      A     M    163.3;
      =     L      4.0;
      BLD   103;
      A     M     21.0;
      =     L      4.1;
      BLD   103;
      A     M     20.1;
      =     L      4.2;
      BLD   103;
      A     M     20.1;
      =     L      4.3;
      BLD   103;
      A     I      8.7;
      =     L      4.4;
      BLD   103;
      A     M     20.0;
      =     L      4.5;
      BLD   103;
      A     M    163.1;
      =     L      4.6;
      BLD   103;
      A     M    163.2;
      =     L      4.7;
      BLD   103;
      CALL FC   180 (
           IN0                      := L      4.0,
           IN1                      := L      4.1,
           IN2                      := L      4.2,
           IN3                      := L      4.3,
           IN4                      := L      4.4,
           IN5                      := L      4.5,
           IN6                      := L      4.6,
           IN7                      := L      4.7,
           IN8                      := W#16#2,
           IN9                      := C      9,
           OUT10                    := DB10.DBW   26,
           OUT11                    := Q      6.3,
           OUT12                    := M    163.4,
           OUT13                    := M    163.5,
           IO14                     := DB181.DBW   18,
           IO15                     := DB10.DBW   60);
      NOP   0;
NETWORK
TITLE =

      A     I      8.7;
      =     L      4.0;
      A     L      4.0;
      BLD   102;
      =     Q      3.6;
      O     L      4.0;
      O     I      1.3;
      =     Q      4.5;
END_FUNCTION

FUNCTION FC 15 : VOID
AUTHOR :
FAMILY : DRIVES
NAME : DRIVES
VERSION : 0.1


VAR_TEMP
  TEMP0 : REAL ;
END_VAR
BEGIN
NETWORK
TITLE =

      A     I      0.2;
      AN    M    164.4;
      A(    ;
      A(    ;
      O     Q      0.0;
      O     I      1.0;
      O     I      2.0;
      O     I      2.2;
      O     I      2.3;
      O     I      2.4;
      O     I      2.6;
      O     I      2.7;
      O(    ;
      A     I      4.1;
      FP    M    218.1;
      )     ;
      )     ;
      =     M    218.0;
      A     M    218.0;
      )     ;
      FP    M    164.0;
      =     M    164.1;
NETWORK
TITLE =

      A(    ;
      A     M     38.0;
      A(    ;
      O     I     11.4;
      O     I     12.5;
      )     ;
      L     DB2.DBW   54;
      SD    T     27;
      NOP   0;
      NOP   0;
      NOP   0;
      A     T     27;
      )     ;
      FP    M    218.3;
      =     M    164.2;
NETWORK
TITLE =
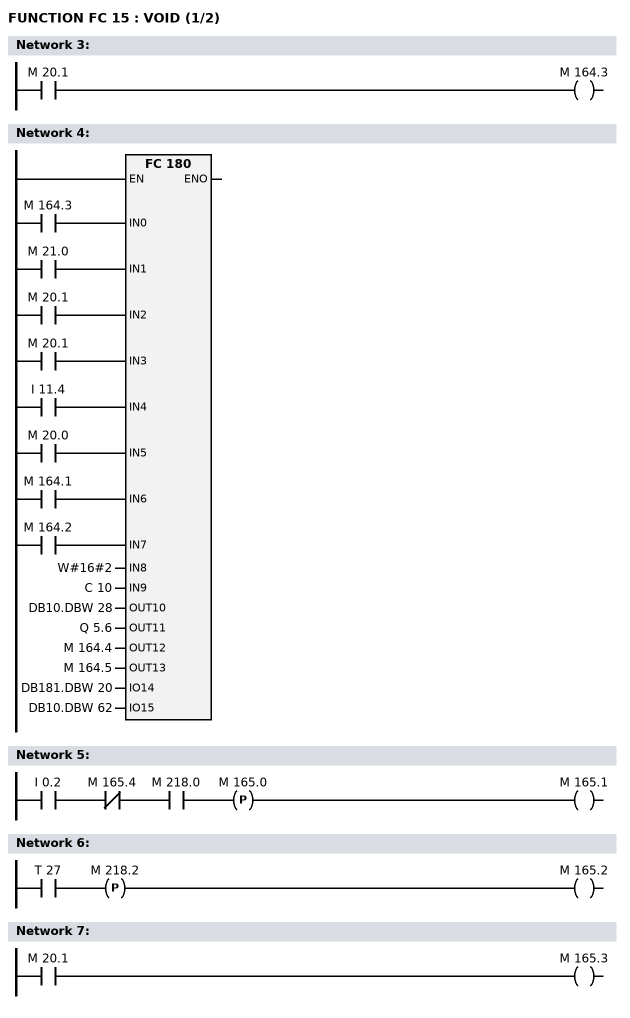

      A     M     20.1;
      =     M    164.3;
NETWORK
TITLE =

      A     M    164.3;
      =     L      4.0;
      BLD   103;
      A     M     21.0;
      =     L      4.1;
      BLD   103;
      A     M     20.1;
      =     L      4.2;
      BLD   103;
      A     M     20.1;
      =     L      4.3;
      BLD   103;
      A     I     11.4;
      =     L      4.4;
      BLD   103;
      A     M     20.0;
      =     L      4.5;
      BLD   103;
      A     M    164.1;
      =     L      4.6;
      BLD   103;
      A     M    164.2;
      =     L      4.7;
      BLD   103;
      CALL FC   180 (
           IN0                      := L      4.0,
           IN1                      := L      4.1,
           IN2                      := L      4.2,
           IN3                      := L      4.3,
           IN4                      := L      4.4,
           IN5                      := L      4.5,
           IN6                      := L      4.6,
           IN7                      := L      4.7,
           IN8                      := W#16#2,
           IN9                      := C     10,
           OUT10                    := DB10.DBW   28,
           OUT11                    := Q      5.6,
           OUT12                    := M    164.4,
           OUT13                    := M    164.5,
           IO14                     := DB181.DBW   20,
           IO15                     := DB10.DBW   62);
      NOP   0;
NETWORK
TITLE =

      A     I      0.2;
      AN    M    165.4;
      A     M    218.0;
      FP    M    165.0;
      =     M    165.1;
NETWORK
TITLE =

      A     T     27;
      FP    M    218.2;
      =     M    165.2;
NETWORK
TITLE =

      A     M     20.1;
      =     M    165.3;
NETWORK
TITLE =
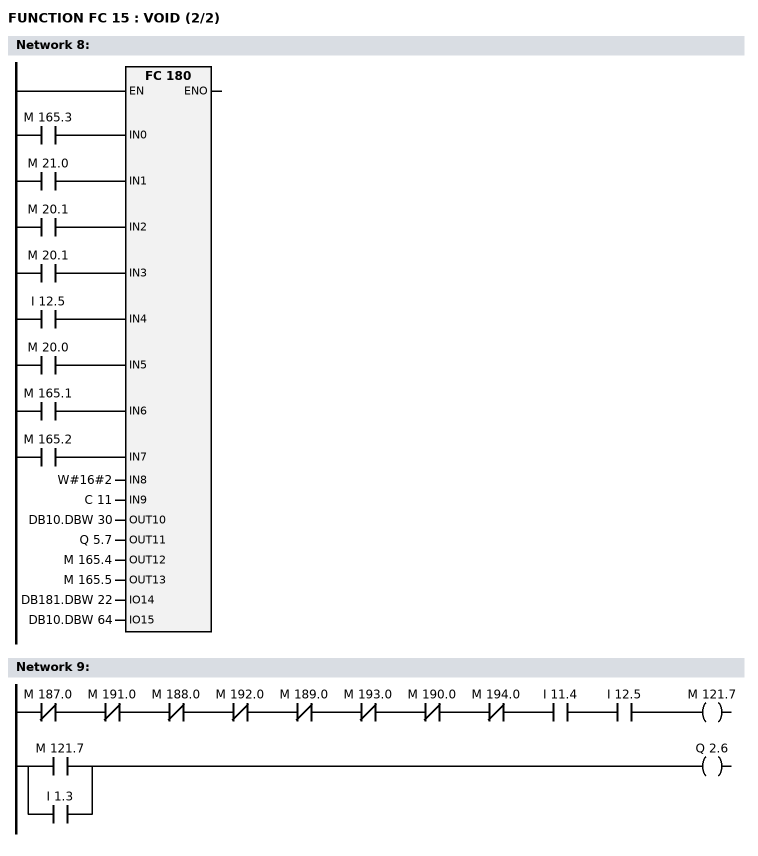

      A     M    165.3;
      =     L      4.0;
      BLD   103;
      A     M     21.0;
      =     L      4.1;
      BLD   103;
      A     M     20.1;
      =     L      4.2;
      BLD   103;
      A     M     20.1;
      =     L      4.3;
      BLD   103;
      A     I     12.5;
      =     L      4.4;
      BLD   103;
      A     M     20.0;
      =     L      4.5;
      BLD   103;
      A     M    165.1;
      =     L      4.6;
      BLD   103;
      A     M    165.2;
      =     L      4.7;
      BLD   103;
      CALL FC   180 (
           IN0                      := L      4.0,
           IN1                      := L      4.1,
           IN2                      := L      4.2,
           IN3                      := L      4.3,
           IN4                      := L      4.4,
           IN5                      := L      4.5,
           IN6                      := L      4.6,
           IN7                      := L      4.7,
           IN8                      := W#16#2,
           IN9                      := C     11,
           OUT10                    := DB10.DBW   30,
           OUT11                    := Q      5.7,
           OUT12                    := M    165.4,
           OUT13                    := M    165.5,
           IO14                     := DB181.DBW   22,
           IO15                     := DB10.DBW   64);
      NOP   0;
NETWORK
TITLE =

      AN    M    187.0;
      AN    M    191.0;
      AN    M    188.0;
      AN    M    192.0;
      AN    M    189.0;
      AN    M    193.0;
      AN    M    190.0;
      AN    M    194.0;
      A     I     11.4;
      A     I     12.5;
      =     M    121.7;
      A     M    121.7;
      O     I      1.3;
      =     Q      2.6;
END_FUNCTION

FUNCTION FC 20 : VOID
AUTHOR :
FAMILY : ANALOGUE
NAME : ANALOGUE
VERSION : 0.1


VAR_TEMP
  TEMP0 : WORD ;
  TEMP1 : REAL ;
  TEMP2 : REAL ;
  TEMP3 : REAL ;
END_VAR
BEGIN
NETWORK
TITLE =
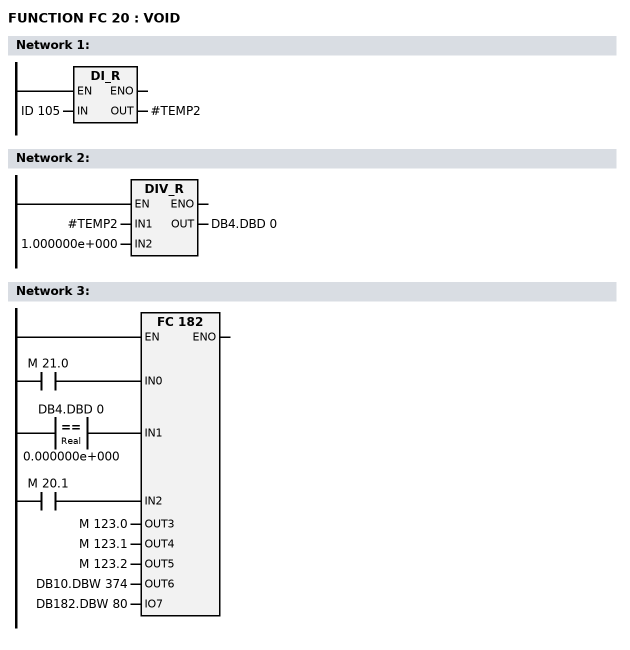

      L     ID   105;
      DTR   ;
      T     #TEMP2;
      NOP   0;
NETWORK
TITLE =

      L     #TEMP2;
      L     1.000000e+000;
      /R    ;
      T     DB4.DBD    0;
      NOP   0;
NETWORK
TITLE =

      A     M     21.0;
      =     L     14.0;
      BLD   103;
      A(    ;
      L     DB4.DBD    0;
      L     0.000000e+000;
      ==R   ;
      )     ;
      =     L     14.1;
      BLD   103;
      A     M     20.1;
      =     L     14.2;
      BLD   103;
      CALL FC   182 (
           IN0                      := L     14.0,
           IN1                      := L     14.1,
           IN2                      := L     14.2,
           OUT3                     := M    123.0,
           OUT4                     := M    123.1,
           OUT5                     := M    123.2,
           OUT6                     := DB10.DBW  374,
           IO7                      := DB182.DBW   80);
      NOP   0;
NETWORK
TITLE =

      A     M    200.6;
      A     M     20.1;
      =     L     14.0;
      A     L     14.0;
      JNB   M001;
      L     DW#16#80000000;
      T     QD   105;
M001: NOP   0;
      AN    L     14.0;
      JNB   M002;
      L     DW#16#0;
      T     QD   105;
M002: NOP   0;
NETWORK
TITLE =

      L     DB4.DBD    0;
      L     DB4.DBD    4;
      >=R   ;
      =     M    116.0;
      =     Q      4.1;
NETWORK
TITLE =

      A(    ;
      L     DB4.DBD    0;
      L     DB4.DBD   12;
      >=R   ;
      )     ;
      A(    ;
      A(    ;
      O     M    116.3;
      O     M    116.5;
      )     ;
      FP    M    122.0;
      )     ;
      S     M    122.1;
      A     Q      6.6;
      R     M    122.1;
      A     M    122.1;
      =     L     14.0;
      A     L     14.0;
      BLD   102;
      =     Q      3.7;
      O     L     14.0;
      O     I      1.3;
      =     Q      1.4;
NETWORK
TITLE =
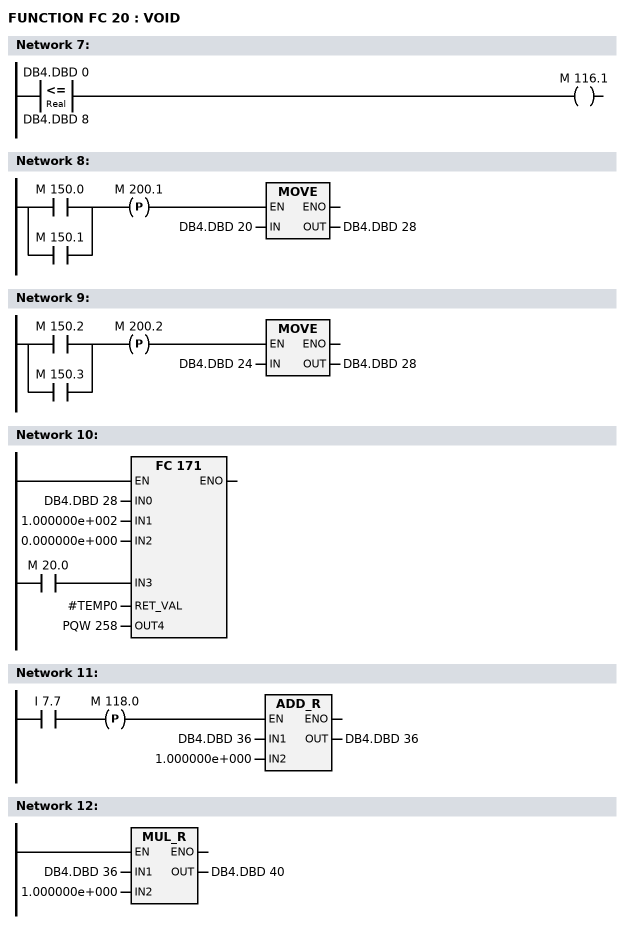

      L     DB4.DBD    0;
      L     DB4.DBD    8;
      <=R   ;
      =     M    116.1;
NETWORK
TITLE =

      A(    ;
      O     M    150.0;
      O     M    150.1;
      )     ;
      FP    M    200.1;
      JNB   M003;
      L     DB4.DBD   20;
      T     DB4.DBD   28;
M003: NOP   0;
NETWORK
TITLE =

      A(    ;
      O     M    150.2;
      O     M    150.3;
      )     ;
      FP    M    200.2;
      JNB   M004;
      L     DB4.DBD   24;
      T     DB4.DBD   28;
M004: NOP   0;
NETWORK
TITLE =

      A     M     20.0;
      =     L     14.0;
      BLD   103;
      CALL FC   171 (
           IN0                      := DB4.DBD   28,
           IN1                      := 1.000000e+002,
           IN2                      := 0.000000e+000,
           IN3                      := L     14.0,
           RET_VAL                  := #TEMP0,
           OUT4                     := PQW  258);
      NOP   0;
NETWORK
TITLE =

      A     I      7.7;
      FP    M    118.0;
      JNB   M005;
      L     DB4.DBD   36;
      L     1.000000e+000;
      +R    ;
      T     DB4.DBD   36;
M005: NOP   0;
NETWORK
TITLE =

      L     DB4.DBD   36;
      L     1.000000e+000;
      *R    ;
      T     DB4.DBD   40;
      NOP   0;
NETWORK
TITLE =

      A(    ;
      A(    ;
      A     M    151.3;
      L     DB2.DBW   40;
      SF    T     20;
      NOP   0;
      NOP   0;
      NOP   0;
      A     T     20;
      )     ;
      A(    ;
      O     M    116.5;
      O     M    116.2;
      )     ;
      O     ;
      A(    ;
      A     M    151.2;
      L     DB2.DBW   42;
      SF    T     21;
      NOP   0;
      NOP   0;
      NOP   0;
      A     T     21;
      )     ;
      A(    ;
      O     M    116.3;
      O     M    116.6;
      )     ;
      )     ;
      FP    M    118.2;
      JNB   M006;
      L     0.000000e+000;
      T     DB4.DBD   36;
M006: NOP   0;
NETWORK
TITLE =
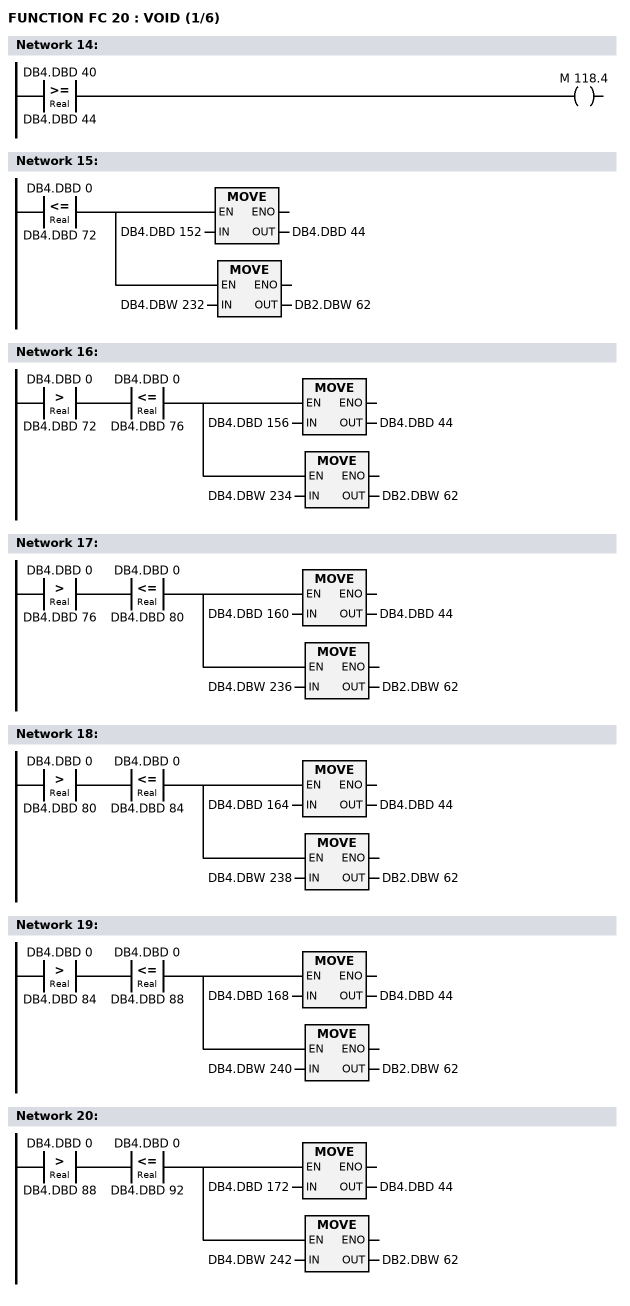

      L     DB4.DBD   40;
      L     DB4.DBD   44;
      >=R   ;
      =     M    118.4;
NETWORK
TITLE =

      L     DB4.DBD    0;
      L     DB4.DBD   72;
      <=R   ;
      =     L     14.0;
      A     L     14.0;
      JNB   M007;
      L     DB4.DBD  152;
      T     DB4.DBD   44;
M007: NOP   0;
      A     L     14.0;
      JNB   M008;
      L     DB4.DBW  232;
      T     DB2.DBW   62;
M008: NOP   0;
NETWORK
TITLE =

      A(    ;
      L     DB4.DBD    0;
      L     DB4.DBD   72;
      >R    ;
      )     ;
      A(    ;
      L     DB4.DBD    0;
      L     DB4.DBD   76;
      <=R   ;
      )     ;
      =     L     14.0;
      A     L     14.0;
      JNB   M009;
      L     DB4.DBD  156;
      T     DB4.DBD   44;
M009: NOP   0;
      A     L     14.0;
      JNB   M00a;
      L     DB4.DBW  234;
      T     DB2.DBW   62;
M00a: NOP   0;
NETWORK
TITLE =

      A(    ;
      L     DB4.DBD    0;
      L     DB4.DBD   76;
      >R    ;
      )     ;
      A(    ;
      L     DB4.DBD    0;
      L     DB4.DBD   80;
      <=R   ;
      )     ;
      =     L     14.0;
      A     L     14.0;
      JNB   M00b;
      L     DB4.DBD  160;
      T     DB4.DBD   44;
M00b: NOP   0;
      A     L     14.0;
      JNB   M00c;
      L     DB4.DBW  236;
      T     DB2.DBW   62;
M00c: NOP   0;
NETWORK
TITLE =

      A(    ;
      L     DB4.DBD    0;
      L     DB4.DBD   80;
      >R    ;
      )     ;
      A(    ;
      L     DB4.DBD    0;
      L     DB4.DBD   84;
      <=R   ;
      )     ;
      =     L     14.0;
      A     L     14.0;
      JNB   M00d;
      L     DB4.DBD  164;
      T     DB4.DBD   44;
M00d: NOP   0;
      A     L     14.0;
      JNB   M00e;
      L     DB4.DBW  238;
      T     DB2.DBW   62;
M00e: NOP   0;
NETWORK
TITLE =

      A(    ;
      L     DB4.DBD    0;
      L     DB4.DBD   84;
      >R    ;
      )     ;
      A(    ;
      L     DB4.DBD    0;
      L     DB4.DBD   88;
      <=R   ;
      )     ;
      =     L     14.0;
      A     L     14.0;
      JNB   M00f;
      L     DB4.DBD  168;
      T     DB4.DBD   44;
M00f: NOP   0;
      A     L     14.0;
      JNB   M010;
      L     DB4.DBW  240;
      T     DB2.DBW   62;
M010: NOP   0;
NETWORK
TITLE =

      A(    ;
      L     DB4.DBD    0;
      L     DB4.DBD   88;
      >R    ;
      )     ;
      A(    ;
      L     DB4.DBD    0;
      L     DB4.DBD   92;
      <=R   ;
      )     ;
      =     L     14.0;
      A     L     14.0;
      JNB   M011;
      L     DB4.DBD  172;
      T     DB4.DBD   44;
M011: NOP   0;
      A     L     14.0;
      JNB   M012;
      L     DB4.DBW  242;
      T     DB2.DBW   62;
M012: NOP   0;
NETWORK
TITLE =
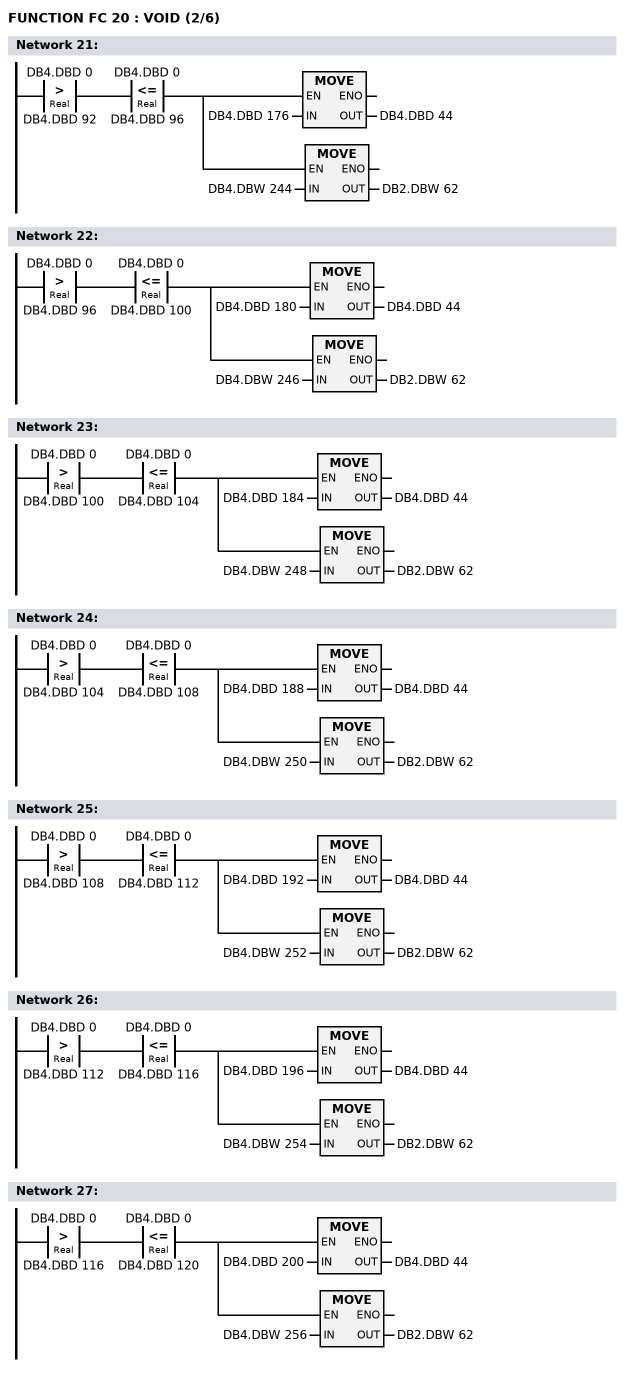

      A(    ;
      L     DB4.DBD    0;
      L     DB4.DBD   92;
      >R    ;
      )     ;
      A(    ;
      L     DB4.DBD    0;
      L     DB4.DBD   96;
      <=R   ;
      )     ;
      =     L     14.0;
      A     L     14.0;
      JNB   M013;
      L     DB4.DBD  176;
      T     DB4.DBD   44;
M013: NOP   0;
      A     L     14.0;
      JNB   M014;
      L     DB4.DBW  244;
      T     DB2.DBW   62;
M014: NOP   0;
NETWORK
TITLE =

      A(    ;
      L     DB4.DBD    0;
      L     DB4.DBD   96;
      >R    ;
      )     ;
      A(    ;
      L     DB4.DBD    0;
      L     DB4.DBD  100;
      <=R   ;
      )     ;
      =     L     14.0;
      A     L     14.0;
      JNB   M015;
      L     DB4.DBD  180;
      T     DB4.DBD   44;
M015: NOP   0;
      A     L     14.0;
      JNB   M016;
      L     DB4.DBW  246;
      T     DB2.DBW   62;
M016: NOP   0;
NETWORK
TITLE =

      A(    ;
      L     DB4.DBD    0;
      L     DB4.DBD  100;
      >R    ;
      )     ;
      A(    ;
      L     DB4.DBD    0;
      L     DB4.DBD  104;
      <=R   ;
      )     ;
      =     L     14.0;
      A     L     14.0;
      JNB   M017;
      L     DB4.DBD  184;
      T     DB4.DBD   44;
M017: NOP   0;
      A     L     14.0;
      JNB   M018;
      L     DB4.DBW  248;
      T     DB2.DBW   62;
M018: NOP   0;
NETWORK
TITLE =

      A(    ;
      L     DB4.DBD    0;
      L     DB4.DBD  104;
      >R    ;
      )     ;
      A(    ;
      L     DB4.DBD    0;
      L     DB4.DBD  108;
      <=R   ;
      )     ;
      =     L     14.0;
      A     L     14.0;
      JNB   M019;
      L     DB4.DBD  188;
      T     DB4.DBD   44;
M019: NOP   0;
      A     L     14.0;
      JNB   M01a;
      L     DB4.DBW  250;
      T     DB2.DBW   62;
M01a: NOP   0;
NETWORK
TITLE =

      A(    ;
      L     DB4.DBD    0;
      L     DB4.DBD  108;
      >R    ;
      )     ;
      A(    ;
      L     DB4.DBD    0;
      L     DB4.DBD  112;
      <=R   ;
      )     ;
      =     L     14.0;
      A     L     14.0;
      JNB   M01b;
      L     DB4.DBD  192;
      T     DB4.DBD   44;
M01b: NOP   0;
      A     L     14.0;
      JNB   M01c;
      L     DB4.DBW  252;
      T     DB2.DBW   62;
M01c: NOP   0;
NETWORK
TITLE =

      A(    ;
      L     DB4.DBD    0;
      L     DB4.DBD  112;
      >R    ;
      )     ;
      A(    ;
      L     DB4.DBD    0;
      L     DB4.DBD  116;
      <=R   ;
      )     ;
      =     L     14.0;
      A     L     14.0;
      JNB   M01d;
      L     DB4.DBD  196;
      T     DB4.DBD   44;
M01d: NOP   0;
      A     L     14.0;
      JNB   M01e;
      L     DB4.DBW  254;
      T     DB2.DBW   62;
M01e: NOP   0;
NETWORK
TITLE =

      A(    ;
      L     DB4.DBD    0;
      L     DB4.DBD  116;
      >R    ;
      )     ;
      A(    ;
      L     DB4.DBD    0;
      L     DB4.DBD  120;
      <=R   ;
      )     ;
      =     L     14.0;
      A     L     14.0;
      JNB   M01f;
      L     DB4.DBD  200;
      T     DB4.DBD   44;
M01f: NOP   0;
      A     L     14.0;
      JNB   M020;
      L     DB4.DBW  256;
      T     DB2.DBW   62;
M020: NOP   0;
NETWORK
TITLE =
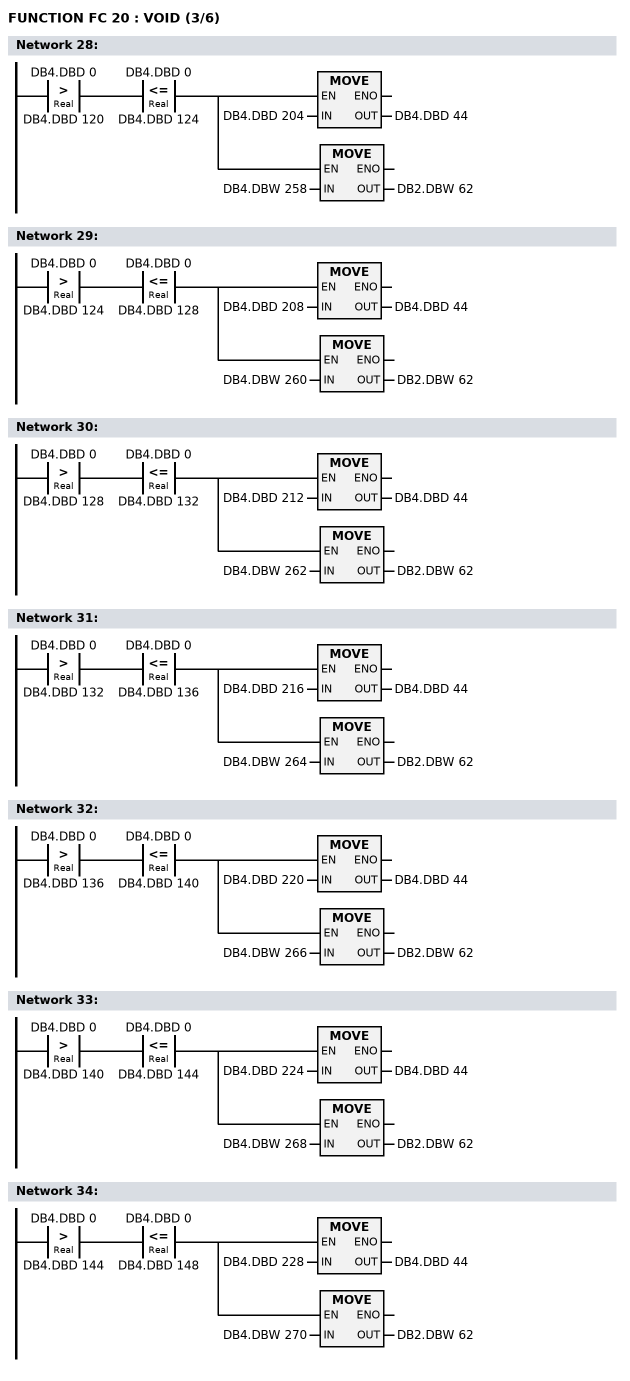

      A(    ;
      L     DB4.DBD    0;
      L     DB4.DBD  120;
      >R    ;
      )     ;
      A(    ;
      L     DB4.DBD    0;
      L     DB4.DBD  124;
      <=R   ;
      )     ;
      =     L     14.0;
      A     L     14.0;
      JNB   M021;
      L     DB4.DBD  204;
      T     DB4.DBD   44;
M021: NOP   0;
      A     L     14.0;
      JNB   M022;
      L     DB4.DBW  258;
      T     DB2.DBW   62;
M022: NOP   0;
NETWORK
TITLE =

      A(    ;
      L     DB4.DBD    0;
      L     DB4.DBD  124;
      >R    ;
      )     ;
      A(    ;
      L     DB4.DBD    0;
      L     DB4.DBD  128;
      <=R   ;
      )     ;
      =     L     14.0;
      A     L     14.0;
      JNB   M023;
      L     DB4.DBD  208;
      T     DB4.DBD   44;
M023: NOP   0;
      A     L     14.0;
      JNB   M024;
      L     DB4.DBW  260;
      T     DB2.DBW   62;
M024: NOP   0;
NETWORK
TITLE =

      A(    ;
      L     DB4.DBD    0;
      L     DB4.DBD  128;
      >R    ;
      )     ;
      A(    ;
      L     DB4.DBD    0;
      L     DB4.DBD  132;
      <=R   ;
      )     ;
      =     L     14.0;
      A     L     14.0;
      JNB   M025;
      L     DB4.DBD  212;
      T     DB4.DBD   44;
M025: NOP   0;
      A     L     14.0;
      JNB   M026;
      L     DB4.DBW  262;
      T     DB2.DBW   62;
M026: NOP   0;
NETWORK
TITLE =

      A(    ;
      L     DB4.DBD    0;
      L     DB4.DBD  132;
      >R    ;
      )     ;
      A(    ;
      L     DB4.DBD    0;
      L     DB4.DBD  136;
      <=R   ;
      )     ;
      =     L     14.0;
      A     L     14.0;
      JNB   M027;
      L     DB4.DBD  216;
      T     DB4.DBD   44;
M027: NOP   0;
      A     L     14.0;
      JNB   M028;
      L     DB4.DBW  264;
      T     DB2.DBW   62;
M028: NOP   0;
NETWORK
TITLE =

      A(    ;
      L     DB4.DBD    0;
      L     DB4.DBD  136;
      >R    ;
      )     ;
      A(    ;
      L     DB4.DBD    0;
      L     DB4.DBD  140;
      <=R   ;
      )     ;
      =     L     14.0;
      A     L     14.0;
      JNB   M029;
      L     DB4.DBD  220;
      T     DB4.DBD   44;
M029: NOP   0;
      A     L     14.0;
      JNB   M02a;
      L     DB4.DBW  266;
      T     DB2.DBW   62;
M02a: NOP   0;
NETWORK
TITLE =

      A(    ;
      L     DB4.DBD    0;
      L     DB4.DBD  140;
      >R    ;
      )     ;
      A(    ;
      L     DB4.DBD    0;
      L     DB4.DBD  144;
      <=R   ;
      )     ;
      =     L     14.0;
      A     L     14.0;
      JNB   M02b;
      L     DB4.DBD  224;
      T     DB4.DBD   44;
M02b: NOP   0;
      A     L     14.0;
      JNB   M02c;
      L     DB4.DBW  268;
      T     DB2.DBW   62;
M02c: NOP   0;
NETWORK
TITLE =

      A(    ;
      L     DB4.DBD    0;
      L     DB4.DBD  144;
      >R    ;
      )     ;
      A(    ;
      L     DB4.DBD    0;
      L     DB4.DBD  148;
      <=R   ;
      )     ;
      =     L     14.0;
      A     L     14.0;
      JNB   M02d;
      L     DB4.DBD  228;
      T     DB4.DBD   44;
M02d: NOP   0;
      A     L     14.0;
      JNB   M02e;
      L     DB4.DBW  270;
      T     DB2.DBW   62;
M02e: NOP   0;
NETWORK
TITLE =
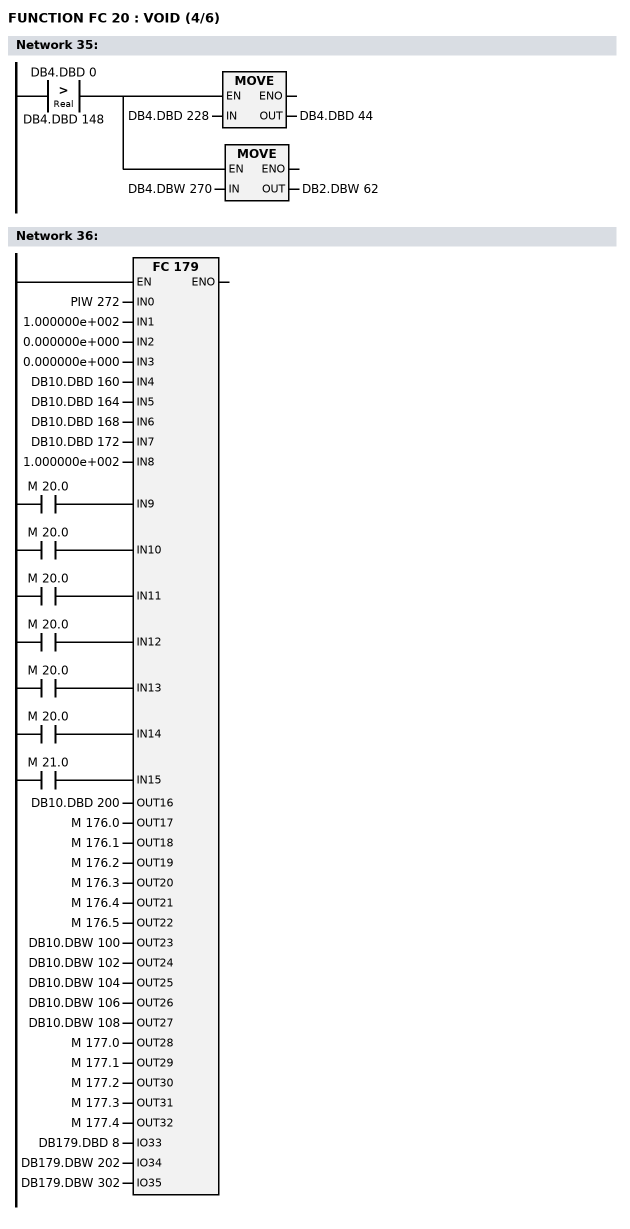

      L     DB4.DBD    0;
      L     DB4.DBD  148;
      >R    ;
      =     L     14.0;
      A     L     14.0;
      JNB   M02f;
      L     DB4.DBD  228;
      T     DB4.DBD   44;
M02f: NOP   0;
      A     L     14.0;
      JNB   M030;
      L     DB4.DBW  270;
      T     DB2.DBW   62;
M030: NOP   0;
NETWORK
TITLE =

      A     M     20.0;
      =     L     14.0;
      BLD   103;
      A     M     20.0;
      =     L     14.1;
      BLD   103;
      A     M     20.0;
      =     L     14.2;
      BLD   103;
      A     M     20.0;
      =     L     14.3;
      BLD   103;
      A     M     20.0;
      =     L     14.4;
      BLD   103;
      A     M     20.0;
      =     L     14.5;
      BLD   103;
      A     M     21.0;
      =     L     14.6;
      BLD   103;
      CALL FC   179 (
           IN0                      := PIW  272,
           IN1                      := 1.000000e+002,
           IN2                      := 0.000000e+000,
           IN3                      := 0.000000e+000,
           IN4                      := DB10.DBD  160,
           IN5                      := DB10.DBD  164,
           IN6                      := DB10.DBD  168,
           IN7                      := DB10.DBD  172,
           IN8                      := 1.000000e+002,
           IN9                      := L     14.0,
           IN10                     := L     14.1,
           IN11                     := L     14.2,
           IN12                     := L     14.3,
           IN13                     := L     14.4,
           IN14                     := L     14.5,
           IN15                     := L     14.6,
           OUT16                    := DB10.DBD  200,
           OUT17                    := M    176.0,
           OUT18                    := M    176.1,
           OUT19                    := M    176.2,
           OUT20                    := M    176.3,
           OUT21                    := M    176.4,
           OUT22                    := M    176.5,
           OUT23                    := DB10.DBW  100,
           OUT24                    := DB10.DBW  102,
           OUT25                    := DB10.DBW  104,
           OUT26                    := DB10.DBW  106,
           OUT27                    := DB10.DBW  108,
           OUT28                    := M    177.0,
           OUT29                    := M    177.1,
           OUT30                    := M    177.2,
           OUT31                    := M    177.3,
           OUT32                    := M    177.4,
           IO33                     := DB179.DBD    8,
           IO34                     := DB179.DBW  202,
           IO35                     := DB179.DBW  302);
      NOP   0;
NETWORK
TITLE =
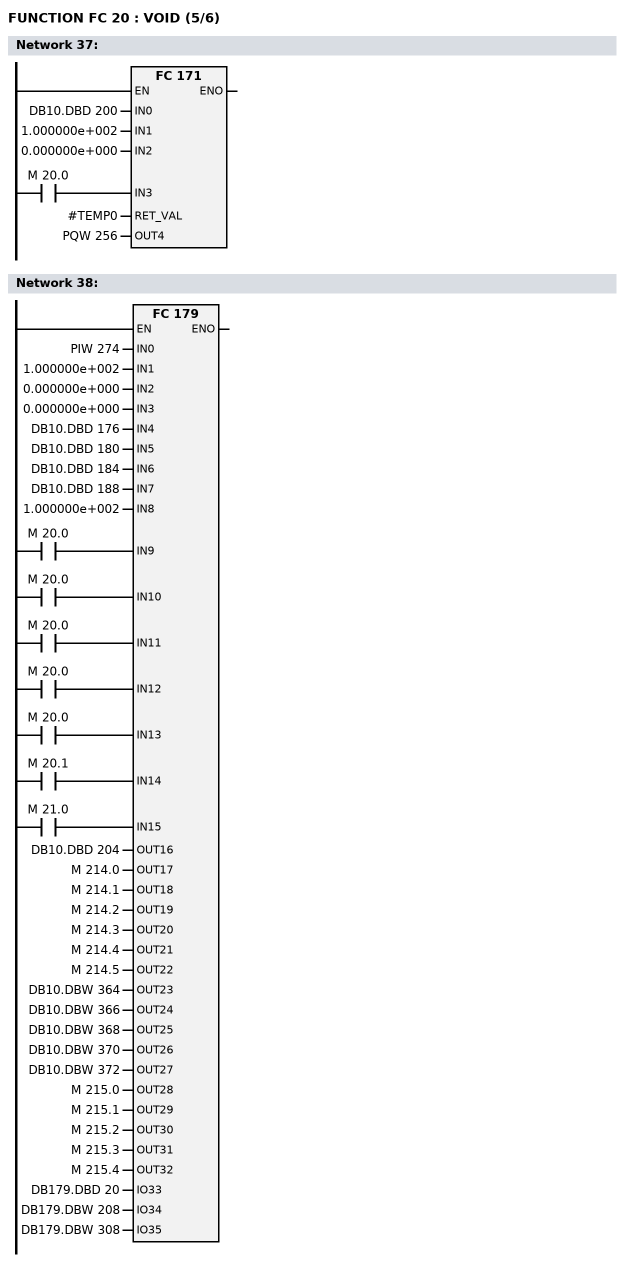

      A     M     20.0;
      =     L     14.0;
      BLD   103;
      CALL FC   171 (
           IN0                      := DB10.DBD  200,
           IN1                      := 1.000000e+002,
           IN2                      := 0.000000e+000,
           IN3                      := L     14.0,
           RET_VAL                  := #TEMP0,
           OUT4                     := PQW  256);
      NOP   0;
NETWORK
TITLE =

      A     M     20.0;
      =     L     14.0;
      BLD   103;
      A     M     20.0;
      =     L     14.1;
      BLD   103;
      A     M     20.0;
      =     L     14.2;
      BLD   103;
      A     M     20.0;
      =     L     14.3;
      BLD   103;
      A     M     20.0;
      =     L     14.4;
      BLD   103;
      A     M     20.1;
      =     L     14.5;
      BLD   103;
      A     M     21.0;
      =     L     14.6;
      BLD   103;
      CALL FC   179 (
           IN0                      := PIW  274,
           IN1                      := 1.000000e+002,
           IN2                      := 0.000000e+000,
           IN3                      := 0.000000e+000,
           IN4                      := DB10.DBD  176,
           IN5                      := DB10.DBD  180,
           IN6                      := DB10.DBD  184,
           IN7                      := DB10.DBD  188,
           IN8                      := 1.000000e+002,
           IN9                      := L     14.0,
           IN10                     := L     14.1,
           IN11                     := L     14.2,
           IN12                     := L     14.3,
           IN13                     := L     14.4,
           IN14                     := L     14.5,
           IN15                     := L     14.6,
           OUT16                    := DB10.DBD  204,
           OUT17                    := M    214.0,
           OUT18                    := M    214.1,
           OUT19                    := M    214.2,
           OUT20                    := M    214.3,
           OUT21                    := M    214.4,
           OUT22                    := M    214.5,
           OUT23                    := DB10.DBW  364,
           OUT24                    := DB10.DBW  366,
           OUT25                    := DB10.DBW  368,
           OUT26                    := DB10.DBW  370,
           OUT27                    := DB10.DBW  372,
           OUT28                    := M    215.0,
           OUT29                    := M    215.1,
           OUT30                    := M    215.2,
           OUT31                    := M    215.3,
           OUT32                    := M    215.4,
           IO33                     := DB179.DBD   20,
           IO34                     := DB179.DBW  208,
           IO35                     := DB179.DBW  308);
      NOP   0;
NETWORK
TITLE =
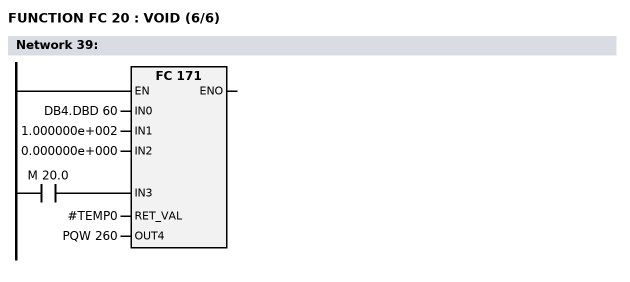

      A     M     20.0;
      =     L     14.0;
      BLD   103;
      CALL FC   171 (
           IN0                      := DB4.DBD   60,
           IN1                      := 1.000000e+002,
           IN2                      := 0.000000e+000,
           IN3                      := L     14.0,
           RET_VAL                  := #TEMP0,
           OUT4                     := PQW  260);
      NOP   0;
END_FUNCTION

FUNCTION FC 21 : VOID
AUTHOR :
FAMILY : DIGITAL
NAME : DIGITAL
VERSION : 0.1


VAR_TEMP
  TEMP0 : WORD ;
END_VAR
BEGIN
NETWORK
TITLE =
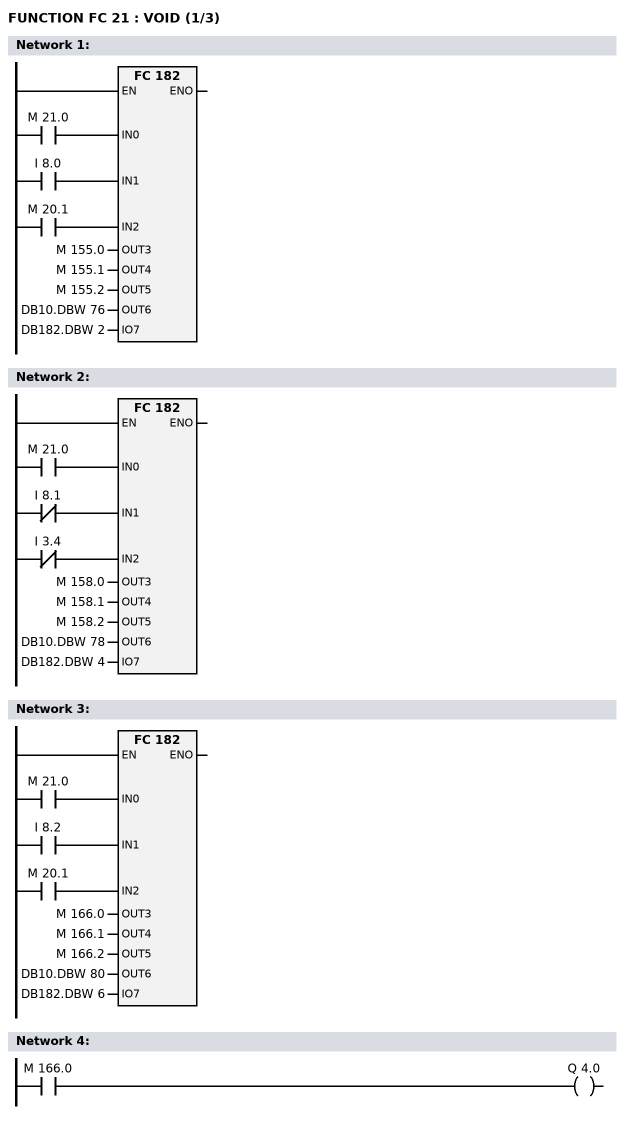

      A     M     21.0;
      =     L      2.0;
      BLD   103;
      A     I      8.0;
      =     L      2.1;
      BLD   103;
      A     M     20.1;
      =     L      2.2;
      BLD   103;
      CALL FC   182 (
           IN0                      := L      2.0,
           IN1                      := L      2.1,
           IN2                      := L      2.2,
           OUT3                     := M    155.0,
           OUT4                     := M    155.1,
           OUT5                     := M    155.2,
           OUT6                     := DB10.DBW   76,
           IO7                      := DB182.DBW    2);
      NOP   0;
NETWORK
TITLE =

      A     M     21.0;
      =     L      2.0;
      BLD   103;
      AN    I      8.1;
      =     L      2.1;
      BLD   103;
      AN    I      3.4;
      =     L      2.2;
      BLD   103;
      CALL FC   182 (
           IN0                      := L      2.0,
           IN1                      := L      2.1,
           IN2                      := L      2.2,
           OUT3                     := M    158.0,
           OUT4                     := M    158.1,
           OUT5                     := M    158.2,
           OUT6                     := DB10.DBW   78,
           IO7                      := DB182.DBW    4);
      NOP   0;
NETWORK
TITLE =

      A     M     21.0;
      =     L      2.0;
      BLD   103;
      A     I      8.2;
      =     L      2.1;
      BLD   103;
      A     M     20.1;
      =     L      2.2;
      BLD   103;
      CALL FC   182 (
           IN0                      := L      2.0,
           IN1                      := L      2.1,
           IN2                      := L      2.2,
           OUT3                     := M    166.0,
           OUT4                     := M    166.1,
           OUT5                     := M    166.2,
           OUT6                     := DB10.DBW   80,
           IO7                      := DB182.DBW    6);
      NOP   0;
NETWORK
TITLE =

      A     M    166.0;
      =     Q      4.0;
NETWORK
TITLE =
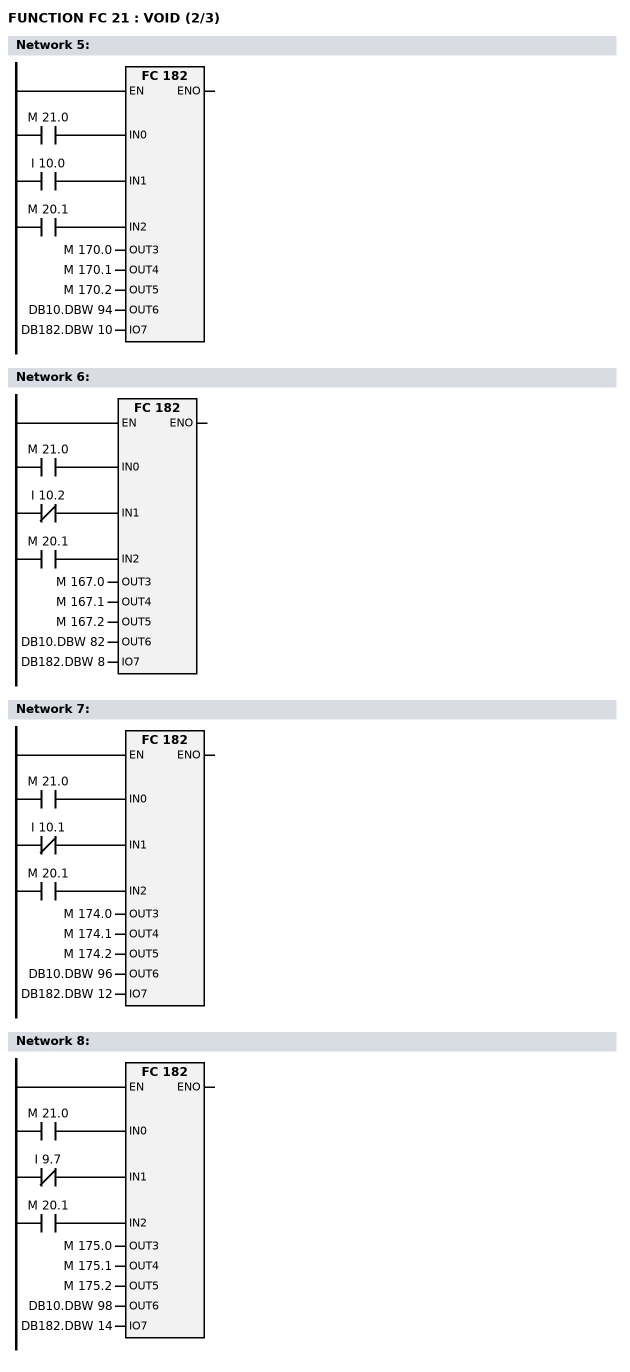

      A     M     21.0;
      =     L      2.0;
      BLD   103;
      A     I     10.0;
      =     L      2.1;
      BLD   103;
      A     M     20.1;
      =     L      2.2;
      BLD   103;
      CALL FC   182 (
           IN0                      := L      2.0,
           IN1                      := L      2.1,
           IN2                      := L      2.2,
           OUT3                     := M    170.0,
           OUT4                     := M    170.1,
           OUT5                     := M    170.2,
           OUT6                     := DB10.DBW   94,
           IO7                      := DB182.DBW   10);
      NOP   0;
NETWORK
TITLE =

      A     M     21.0;
      =     L      2.0;
      BLD   103;
      AN    I     10.2;
      =     L      2.1;
      BLD   103;
      A     M     20.1;
      =     L      2.2;
      BLD   103;
      CALL FC   182 (
           IN0                      := L      2.0,
           IN1                      := L      2.1,
           IN2                      := L      2.2,
           OUT3                     := M    167.0,
           OUT4                     := M    167.1,
           OUT5                     := M    167.2,
           OUT6                     := DB10.DBW   82,
           IO7                      := DB182.DBW    8);
      NOP   0;
NETWORK
TITLE =

      A     M     21.0;
      =     L      2.0;
      BLD   103;
      AN    I     10.1;
      =     L      2.1;
      BLD   103;
      A     M     20.1;
      =     L      2.2;
      BLD   103;
      CALL FC   182 (
           IN0                      := L      2.0,
           IN1                      := L      2.1,
           IN2                      := L      2.2,
           OUT3                     := M    174.0,
           OUT4                     := M    174.1,
           OUT5                     := M    174.2,
           OUT6                     := DB10.DBW   96,
           IO7                      := DB182.DBW   12);
      NOP   0;
NETWORK
TITLE =

      A     M     21.0;
      =     L      2.0;
      BLD   103;
      AN    I      9.7;
      =     L      2.1;
      BLD   103;
      A     M     20.1;
      =     L      2.2;
      BLD   103;
      CALL FC   182 (
           IN0                      := L      2.0,
           IN1                      := L      2.1,
           IN2                      := L      2.2,
           OUT3                     := M    175.0,
           OUT4                     := M    175.1,
           OUT5                     := M    175.2,
           OUT6                     := DB10.DBW   98,
           IO7                      := DB182.DBW   14);
      NOP   0;
NETWORK
TITLE =
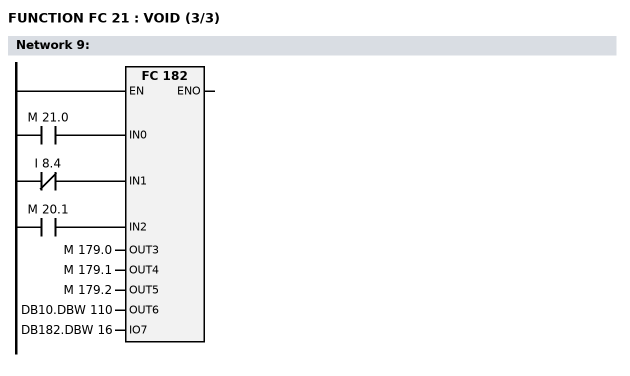

      A     M     21.0;
      =     L      2.0;
      BLD   103;
      AN    I      8.4;
      =     L      2.1;
      BLD   103;
      A     M     20.1;
      =     L      2.2;
      BLD   103;
      CALL FC   182 (
           IN0                      := L      2.0,
           IN1                      := L      2.1,
           IN2                      := L      2.2,
           OUT3                     := M    179.0,
           OUT4                     := M    179.1,
           OUT5                     := M    179.2,
           OUT6                     := DB10.DBW  110,
           IO7                      := DB182.DBW   16);
      NOP   0;
NETWORK
TITLE =

      A     M     21.0;
      =     L      2.0;
      BLD   103;
      AN    I      8.5;
      =     L      2.1;
      BLD   103;
      A(    ;
      A     Q      6.0;
      AN    I      8.5;
      L     DB2.DBW   66;
      SD    T     33;
      NOP   0;
      NOP   0;
      NOP   0;
      A     T     33;
      )     ;
      =     L      2.2;
      BLD   103;
      CALL FC   182 (
           IN0                      := L      2.0,
           IN1                      := L      2.1,
           IN2                      := L      2.2,
           OUT3                     := M    180.0,
           OUT4                     := M    180.1,
           OUT5                     := M    180.2,
           OUT6                     := DB10.DBW  112,
           IO7                      := DB182.DBW   18);
      NOP   0;
NETWORK
TITLE =

      A     M     21.0;
      =     L      2.0;
      BLD   103;
      AN    I      8.6;
      =     L      2.1;
      BLD   103;
      A(    ;
      A     I      8.7;
      L     DB2.DBW   36;
      SD    T     18;
      NOP   0;
      NOP   0;
      NOP   0;
      A     T     18;
      )     ;
      =     L      2.2;
      BLD   103;
      CALL FC   182 (
           IN0                      := L      2.0,
           IN1                      := L      2.1,
           IN2                      := L      2.2,
           OUT3                     := M    181.0,
           OUT4                     := M    181.1,
           OUT5                     := M    181.2,
           OUT6                     := DB10.DBW  310,
           IO7                      := DB182.DBW   20);
      NOP   0;
NETWORK
TITLE =
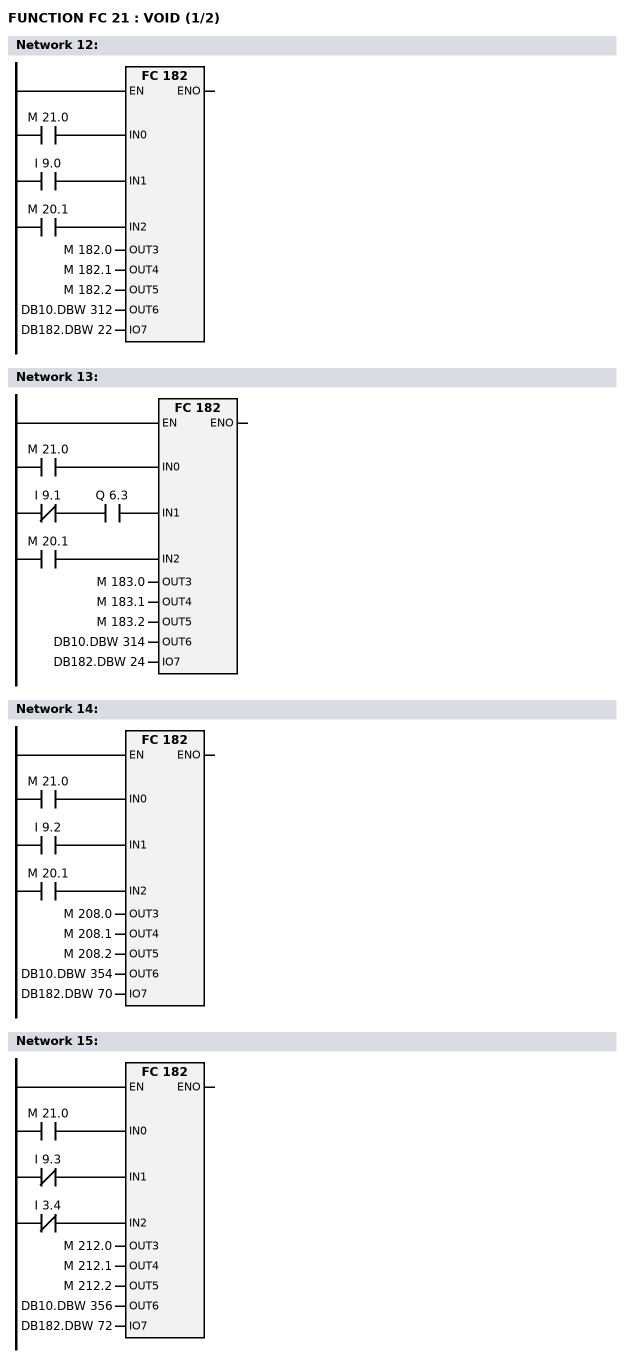

      A     M     21.0;
      =     L      2.0;
      BLD   103;
      A     I      9.0;
      =     L      2.1;
      BLD   103;
      A     M     20.1;
      =     L      2.2;
      BLD   103;
      CALL FC   182 (
           IN0                      := L      2.0,
           IN1                      := L      2.1,
           IN2                      := L      2.2,
           OUT3                     := M    182.0,
           OUT4                     := M    182.1,
           OUT5                     := M    182.2,
           OUT6                     := DB10.DBW  312,
           IO7                      := DB182.DBW   22);
      NOP   0;
NETWORK
TITLE =

      A     M     21.0;
      =     L      2.0;
      BLD   103;
      AN    I      9.1;
      A     Q      6.3;
      =     L      2.1;
      BLD   103;
      A     M     20.1;
      =     L      2.2;
      BLD   103;
      CALL FC   182 (
           IN0                      := L      2.0,
           IN1                      := L      2.1,
           IN2                      := L      2.2,
           OUT3                     := M    183.0,
           OUT4                     := M    183.1,
           OUT5                     := M    183.2,
           OUT6                     := DB10.DBW  314,
           IO7                      := DB182.DBW   24);
      NOP   0;
NETWORK
TITLE =

      A     M     21.0;
      =     L      2.0;
      BLD   103;
      A     I      9.2;
      =     L      2.1;
      BLD   103;
      A     M     20.1;
      =     L      2.2;
      BLD   103;
      CALL FC   182 (
           IN0                      := L      2.0,
           IN1                      := L      2.1,
           IN2                      := L      2.2,
           OUT3                     := M    208.0,
           OUT4                     := M    208.1,
           OUT5                     := M    208.2,
           OUT6                     := DB10.DBW  354,
           IO7                      := DB182.DBW   70);
      NOP   0;
NETWORK
TITLE =

      A     M     21.0;
      =     L      2.0;
      BLD   103;
      AN    I      9.3;
      =     L      2.1;
      BLD   103;
      AN    I      3.4;
      =     L      2.2;
      BLD   103;
      CALL FC   182 (
           IN0                      := L      2.0,
           IN1                      := L      2.1,
           IN2                      := L      2.2,
           OUT3                     := M    212.0,
           OUT4                     := M    212.1,
           OUT5                     := M    212.2,
           OUT6                     := DB10.DBW  356,
           IO7                      := DB182.DBW   72);
      NOP   0;
NETWORK
TITLE =
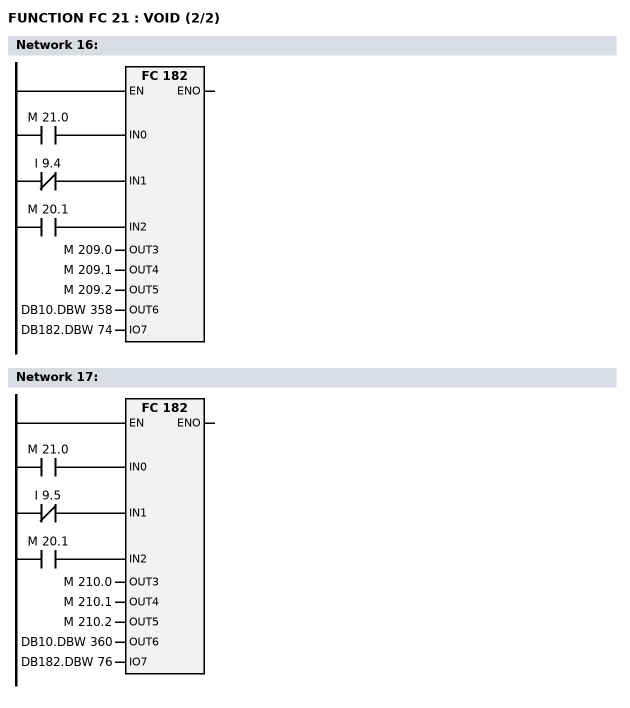

      A     M     21.0;
      =     L      2.0;
      BLD   103;
      AN    I      9.4;
      =     L      2.1;
      BLD   103;
      A     M     20.1;
      =     L      2.2;
      BLD   103;
      CALL FC   182 (
           IN0                      := L      2.0,
           IN1                      := L      2.1,
           IN2                      := L      2.2,
           OUT3                     := M    209.0,
           OUT4                     := M    209.1,
           OUT5                     := M    209.2,
           OUT6                     := DB10.DBW  358,
           IO7                      := DB182.DBW   74);
      NOP   0;
NETWORK
TITLE =

      A     M     21.0;
      =     L      2.0;
      BLD   103;
      AN    I      9.5;
      =     L      2.1;
      BLD   103;
      A     M     20.1;
      =     L      2.2;
      BLD   103;
      CALL FC   182 (
           IN0                      := L      2.0,
           IN1                      := L      2.1,
           IN2                      := L      2.2,
           OUT3                     := M    210.0,
           OUT4                     := M    210.1,
           OUT5                     := M    210.2,
           OUT6                     := DB10.DBW  360,
           IO7                      := DB182.DBW   76);
      NOP   0;
NETWORK
TITLE =

      A     M     21.0;
      =     L      2.0;
      BLD   103;
      A(    ;
      AN    I      9.6;
      A     I      8.7;
      L     DB2.DBW   84;
      SD    T     42;
      NOP   0;
      NOP   0;
      NOP   0;
      A     T     42;
      )     ;
      =     L      2.1;
      BLD   103;
      A     M     20.1;
      =     L      2.2;
      BLD   103;
      CALL FC   182 (
           IN0                      := L      2.0,
           IN1                      := L      2.1,
           IN2                      := L      2.2,
           OUT3                     := M    211.0,
           OUT4                     := M    211.1,
           OUT5                     := M    211.2,
           OUT6                     := DB10.DBW  362,
           IO7                      := DB182.DBW   78);
      NOP   0;
NETWORK
TITLE =
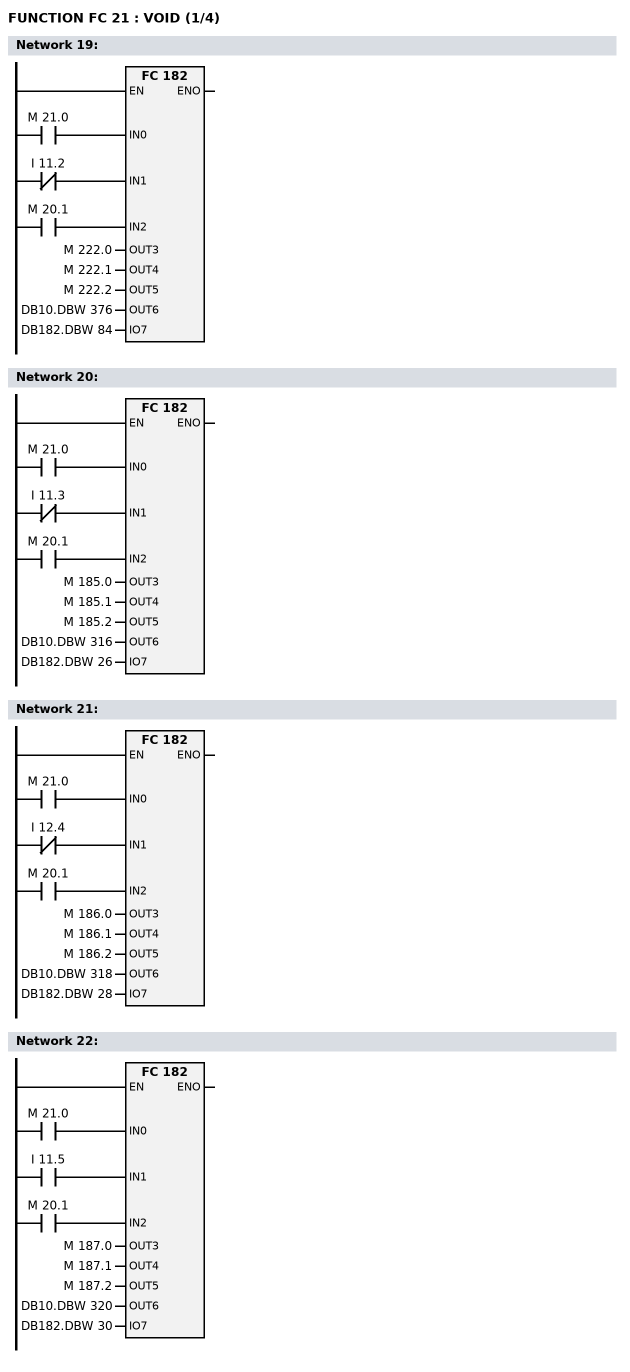

      A     M     21.0;
      =     L      2.0;
      BLD   103;
      AN    I     11.2;
      =     L      2.1;
      BLD   103;
      A     M     20.1;
      =     L      2.2;
      BLD   103;
      CALL FC   182 (
           IN0                      := L      2.0,
           IN1                      := L      2.1,
           IN2                      := L      2.2,
           OUT3                     := M    222.0,
           OUT4                     := M    222.1,
           OUT5                     := M    222.2,
           OUT6                     := DB10.DBW  376,
           IO7                      := DB182.DBW   84);
      NOP   0;
NETWORK
TITLE =

      A     M     21.0;
      =     L      2.0;
      BLD   103;
      AN    I     11.3;
      =     L      2.1;
      BLD   103;
      A     M     20.1;
      =     L      2.2;
      BLD   103;
      CALL FC   182 (
           IN0                      := L      2.0,
           IN1                      := L      2.1,
           IN2                      := L      2.2,
           OUT3                     := M    185.0,
           OUT4                     := M    185.1,
           OUT5                     := M    185.2,
           OUT6                     := DB10.DBW  316,
           IO7                      := DB182.DBW   26);
      NOP   0;
NETWORK
TITLE =

      A     M     21.0;
      =     L      2.0;
      BLD   103;
      AN    I     12.4;
      =     L      2.1;
      BLD   103;
      A     M     20.1;
      =     L      2.2;
      BLD   103;
      CALL FC   182 (
           IN0                      := L      2.0,
           IN1                      := L      2.1,
           IN2                      := L      2.2,
           OUT3                     := M    186.0,
           OUT4                     := M    186.1,
           OUT5                     := M    186.2,
           OUT6                     := DB10.DBW  318,
           IO7                      := DB182.DBW   28);
      NOP   0;
NETWORK
TITLE =

      A     M     21.0;
      =     L      2.0;
      BLD   103;
      A     I     11.5;
      =     L      2.1;
      BLD   103;
      A     M     20.1;
      =     L      2.2;
      BLD   103;
      CALL FC   182 (
           IN0                      := L      2.0,
           IN1                      := L      2.1,
           IN2                      := L      2.2,
           OUT3                     := M    187.0,
           OUT4                     := M    187.1,
           OUT5                     := M    187.2,
           OUT6                     := DB10.DBW  320,
           IO7                      := DB182.DBW   30);
      NOP   0;
NETWORK
TITLE =
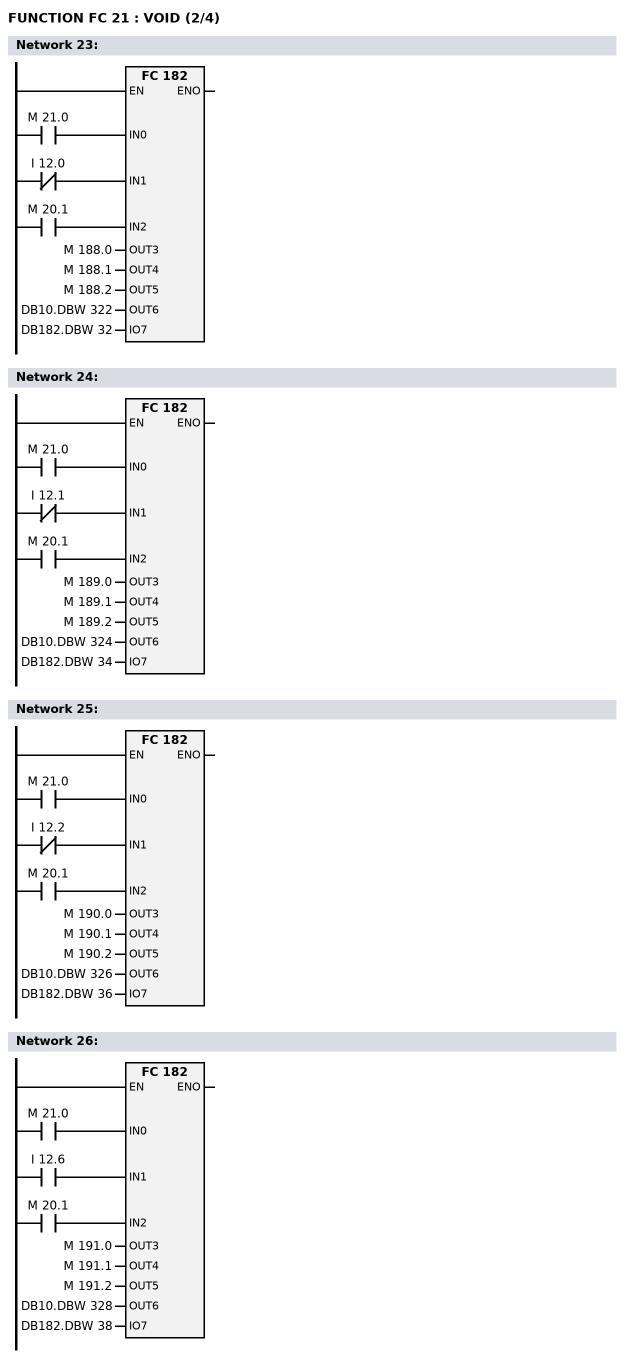

      A     M     21.0;
      =     L      2.0;
      BLD   103;
      AN    I     12.0;
      =     L      2.1;
      BLD   103;
      A     M     20.1;
      =     L      2.2;
      BLD   103;
      CALL FC   182 (
           IN0                      := L      2.0,
           IN1                      := L      2.1,
           IN2                      := L      2.2,
           OUT3                     := M    188.0,
           OUT4                     := M    188.1,
           OUT5                     := M    188.2,
           OUT6                     := DB10.DBW  322,
           IO7                      := DB182.DBW   32);
      NOP   0;
NETWORK
TITLE =

      A     M     21.0;
      =     L      2.0;
      BLD   103;
      AN    I     12.1;
      =     L      2.1;
      BLD   103;
      A     M     20.1;
      =     L      2.2;
      BLD   103;
      CALL FC   182 (
           IN0                      := L      2.0,
           IN1                      := L      2.1,
           IN2                      := L      2.2,
           OUT3                     := M    189.0,
           OUT4                     := M    189.1,
           OUT5                     := M    189.2,
           OUT6                     := DB10.DBW  324,
           IO7                      := DB182.DBW   34);
      NOP   0;
NETWORK
TITLE =

      A     M     21.0;
      =     L      2.0;
      BLD   103;
      AN    I     12.2;
      =     L      2.1;
      BLD   103;
      A     M     20.1;
      =     L      2.2;
      BLD   103;
      CALL FC   182 (
           IN0                      := L      2.0,
           IN1                      := L      2.1,
           IN2                      := L      2.2,
           OUT3                     := M    190.0,
           OUT4                     := M    190.1,
           OUT5                     := M    190.2,
           OUT6                     := DB10.DBW  326,
           IO7                      := DB182.DBW   36);
      NOP   0;
NETWORK
TITLE =

      A     M     21.0;
      =     L      2.0;
      BLD   103;
      A     I     12.6;
      =     L      2.1;
      BLD   103;
      A     M     20.1;
      =     L      2.2;
      BLD   103;
      CALL FC   182 (
           IN0                      := L      2.0,
           IN1                      := L      2.1,
           IN2                      := L      2.2,
           OUT3                     := M    191.0,
           OUT4                     := M    191.1,
           OUT5                     := M    191.2,
           OUT6                     := DB10.DBW  328,
           IO7                      := DB182.DBW   38);
      NOP   0;
NETWORK
TITLE =
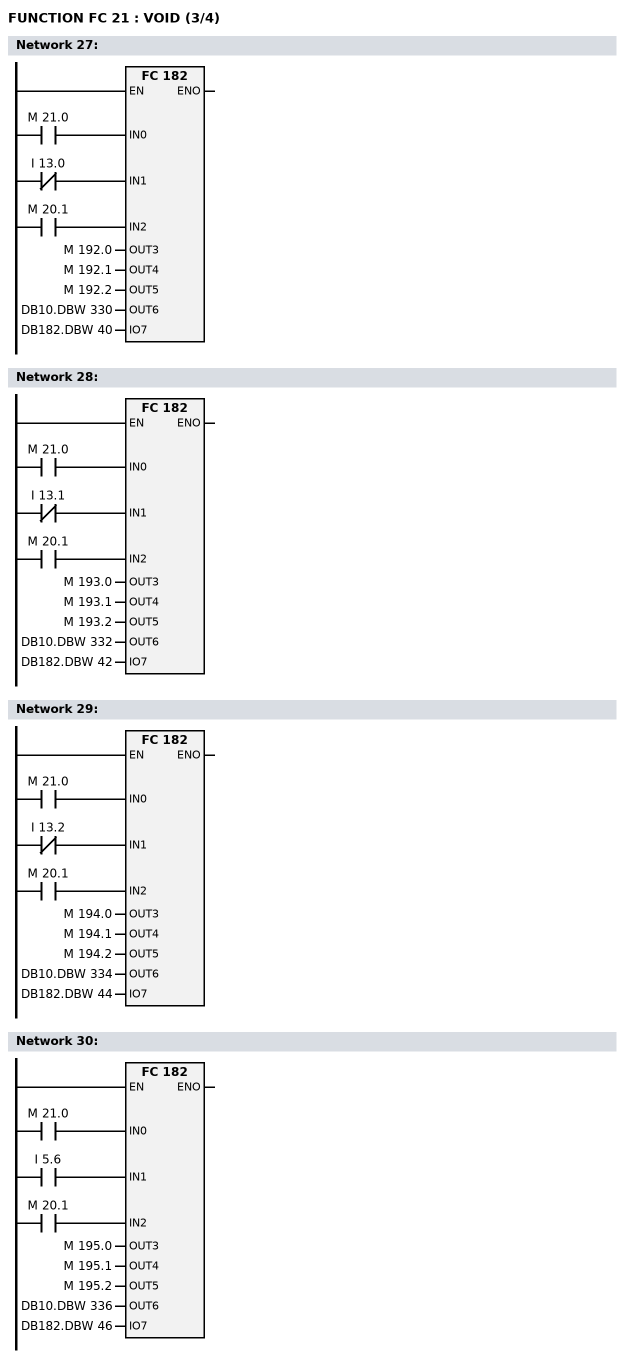

      A     M     21.0;
      =     L      2.0;
      BLD   103;
      AN    I     13.0;
      =     L      2.1;
      BLD   103;
      A     M     20.1;
      =     L      2.2;
      BLD   103;
      CALL FC   182 (
           IN0                      := L      2.0,
           IN1                      := L      2.1,
           IN2                      := L      2.2,
           OUT3                     := M    192.0,
           OUT4                     := M    192.1,
           OUT5                     := M    192.2,
           OUT6                     := DB10.DBW  330,
           IO7                      := DB182.DBW   40);
      NOP   0;
NETWORK
TITLE =

      A     M     21.0;
      =     L      2.0;
      BLD   103;
      AN    I     13.1;
      =     L      2.1;
      BLD   103;
      A     M     20.1;
      =     L      2.2;
      BLD   103;
      CALL FC   182 (
           IN0                      := L      2.0,
           IN1                      := L      2.1,
           IN2                      := L      2.2,
           OUT3                     := M    193.0,
           OUT4                     := M    193.1,
           OUT5                     := M    193.2,
           OUT6                     := DB10.DBW  332,
           IO7                      := DB182.DBW   42);
      NOP   0;
NETWORK
TITLE =

      A     M     21.0;
      =     L      2.0;
      BLD   103;
      AN    I     13.2;
      =     L      2.1;
      BLD   103;
      A     M     20.1;
      =     L      2.2;
      BLD   103;
      CALL FC   182 (
           IN0                      := L      2.0,
           IN1                      := L      2.1,
           IN2                      := L      2.2,
           OUT3                     := M    194.0,
           OUT4                     := M    194.1,
           OUT5                     := M    194.2,
           OUT6                     := DB10.DBW  334,
           IO7                      := DB182.DBW   44);
      NOP   0;
NETWORK
TITLE =

      A     M     21.0;
      =     L      2.0;
      BLD   103;
      A     I      5.6;
      =     L      2.1;
      BLD   103;
      A     M     20.1;
      =     L      2.2;
      BLD   103;
      CALL FC   182 (
           IN0                      := L      2.0,
           IN1                      := L      2.1,
           IN2                      := L      2.2,
           OUT3                     := M    195.0,
           OUT4                     := M    195.1,
           OUT5                     := M    195.2,
           OUT6                     := DB10.DBW  336,
           IO7                      := DB182.DBW   46);
      NOP   0;
NETWORK
TITLE =
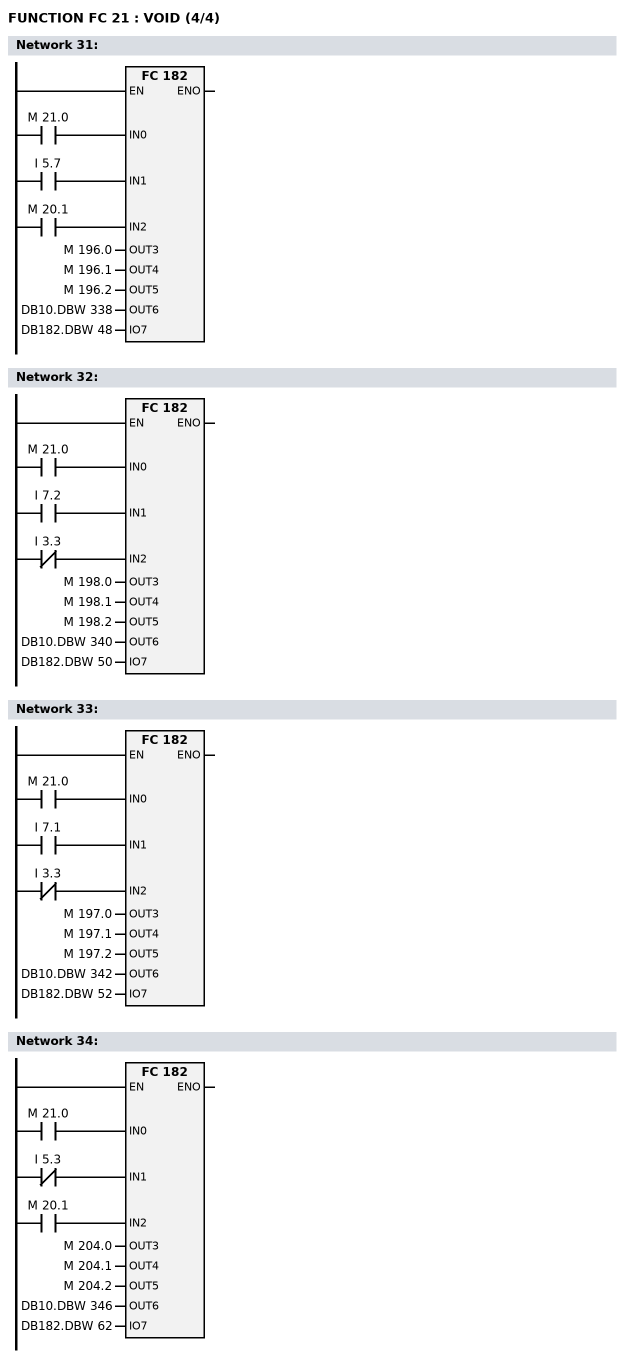

      A     M     21.0;
      =     L      2.0;
      BLD   103;
      A     I      5.7;
      =     L      2.1;
      BLD   103;
      A     M     20.1;
      =     L      2.2;
      BLD   103;
      CALL FC   182 (
           IN0                      := L      2.0,
           IN1                      := L      2.1,
           IN2                      := L      2.2,
           OUT3                     := M    196.0,
           OUT4                     := M    196.1,
           OUT5                     := M    196.2,
           OUT6                     := DB10.DBW  338,
           IO7                      := DB182.DBW   48);
      NOP   0;
NETWORK
TITLE =

      A     M     21.0;
      =     L      2.0;
      BLD   103;
      A     I      7.2;
      =     L      2.1;
      BLD   103;
      AN    I      3.3;
      =     L      2.2;
      BLD   103;
      CALL FC   182 (
           IN0                      := L      2.0,
           IN1                      := L      2.1,
           IN2                      := L      2.2,
           OUT3                     := M    198.0,
           OUT4                     := M    198.1,
           OUT5                     := M    198.2,
           OUT6                     := DB10.DBW  340,
           IO7                      := DB182.DBW   50);
      NOP   0;
NETWORK
TITLE =

      A     M     21.0;
      =     L      2.0;
      BLD   103;
      A     I      7.1;
      =     L      2.1;
      BLD   103;
      AN    I      3.3;
      =     L      2.2;
      BLD   103;
      CALL FC   182 (
           IN0                      := L      2.0,
           IN1                      := L      2.1,
           IN2                      := L      2.2,
           OUT3                     := M    197.0,
           OUT4                     := M    197.1,
           OUT5                     := M    197.2,
           OUT6                     := DB10.DBW  342,
           IO7                      := DB182.DBW   52);
      NOP   0;
NETWORK
TITLE =

      A     M     21.0;
      =     L      2.0;
      BLD   103;
      AN    I      5.3;
      =     L      2.1;
      BLD   103;
      A     M     20.1;
      =     L      2.2;
      BLD   103;
      CALL FC   182 (
           IN0                      := L      2.0,
           IN1                      := L      2.1,
           IN2                      := L      2.2,
           OUT3                     := M    204.0,
           OUT4                     := M    204.1,
           OUT5                     := M    204.2,
           OUT6                     := DB10.DBW  346,
           IO7                      := DB182.DBW   62);
      NOP   0;
NETWORK
TITLE =

      A     M     21.0;
      =     L      2.0;
      BLD   103;
      A(    ;
      A(    ;
      O     Q      6.0;
      O     Q      6.1;
      )     ;
      L     DB2.DBW   50;
      SD    T     25;
      NOP   0;
      NOP   0;
      NOP   0;
      A     T     25;
      )     ;
      A(    ;
      ON    I      6.0;
      ON    I      6.1;
      )     ;
      =     M    216.0;
      A     M    216.0;
      =     L      2.1;
      BLD   103;
      A     M     20.1;
      =     L      2.2;
      BLD   103;
      CALL FC   182 (
           IN0                      := L      2.0,
           IN1                      := L      2.1,
           IN2                      := L      2.2,
           OUT3                     := M    217.0,
           OUT4                     := M    217.1,
           OUT5                     := M    217.2,
           OUT6                     := DB10.DBW  348,
           IO7                      := DB182.DBW   82);
      NOP   0;
END_FUNCTION

FUNCTION FC 3 : VOID
AUTHOR :
FAMILY : Alarm
NAME : Alarm
VERSION : 0.1

BEGIN
NETWORK
TITLE =
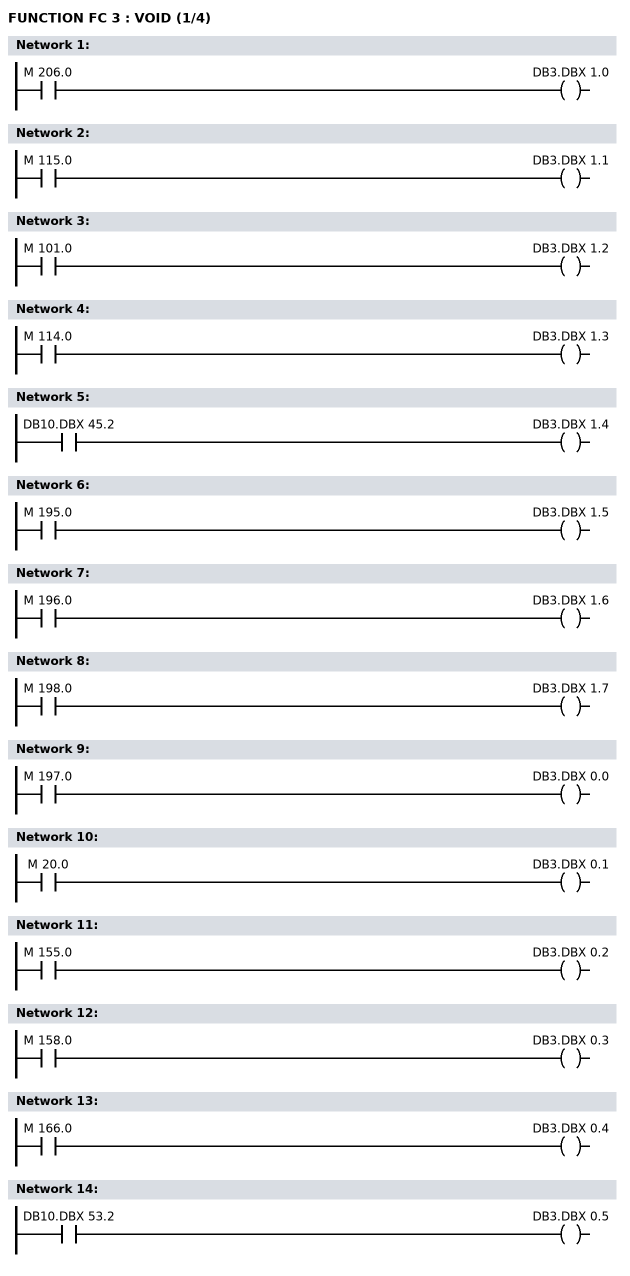

      A     M    206.0;
      =     DB3.DBX    1.0;
NETWORK
TITLE =

      A     M    115.0;
      =     DB3.DBX    1.1;
NETWORK
TITLE =

      A     M    101.0;
      =     DB3.DBX    1.2;
NETWORK
TITLE =

      A     M    114.0;
      =     DB3.DBX    1.3;
NETWORK
TITLE =

      A     DB10.DBX   45.2;
      =     DB3.DBX    1.4;
NETWORK
TITLE =

      A     M    195.0;
      =     DB3.DBX    1.5;
NETWORK
TITLE =

      A     M    196.0;
      =     DB3.DBX    1.6;
NETWORK
TITLE =

      A     M    198.0;
      =     DB3.DBX    1.7;
NETWORK
TITLE =

      A     M    197.0;
      =     DB3.DBX    0.0;
NETWORK
TITLE =

      A     M     20.0;
      =     DB3.DBX    0.1;
NETWORK
TITLE =

      A     M    155.0;
      =     DB3.DBX    0.2;
NETWORK
TITLE =

      A     M    158.0;
      =     DB3.DBX    0.3;
NETWORK
TITLE =

      A     M    166.0;
      =     DB3.DBX    0.4;
NETWORK
TITLE =

      A     DB10.DBX   53.2;
      =     DB3.DBX    0.5;
NETWORK
TITLE =
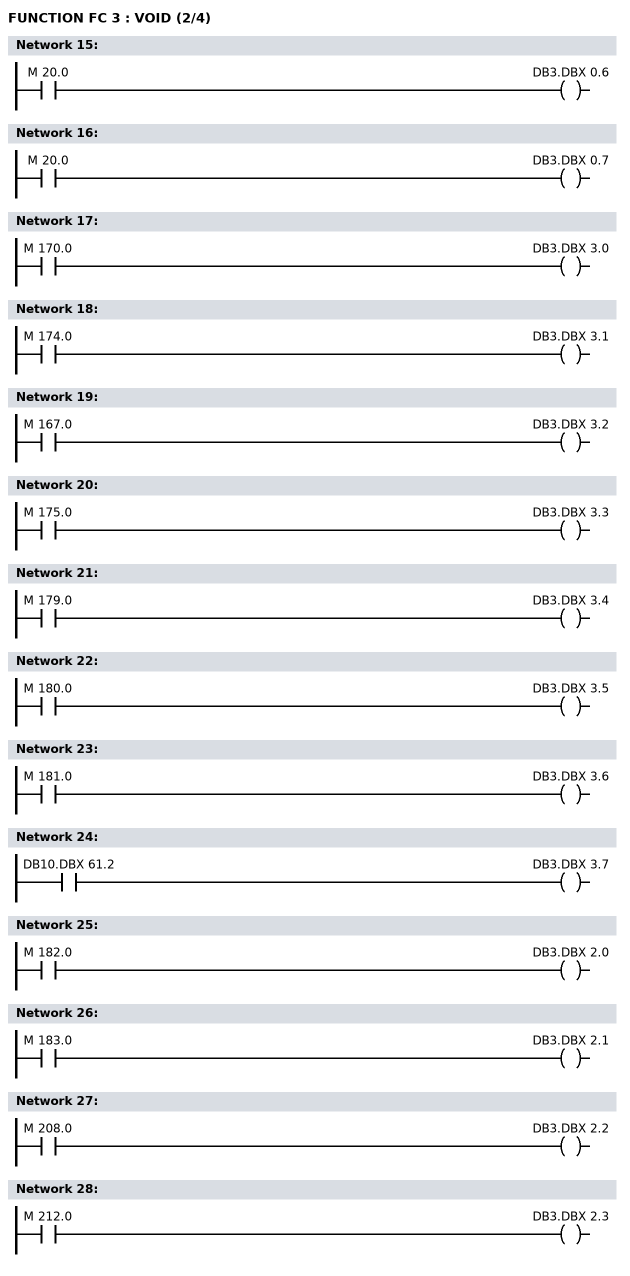

      A     M     20.0;
      =     DB3.DBX    0.6;
NETWORK
TITLE =

      A     M     20.0;
      =     DB3.DBX    0.7;
NETWORK
TITLE =

      A     M    170.0;
      =     DB3.DBX    3.0;
NETWORK
TITLE =

      A     M    174.0;
      =     DB3.DBX    3.1;
NETWORK
TITLE =

      A     M    167.0;
      =     DB3.DBX    3.2;
NETWORK
TITLE =

      A     M    175.0;
      =     DB3.DBX    3.3;
NETWORK
TITLE =

      A     M    179.0;
      =     DB3.DBX    3.4;
NETWORK
TITLE =

      A     M    180.0;
      =     DB3.DBX    3.5;
NETWORK
TITLE =

      A     M    181.0;
      =     DB3.DBX    3.6;
NETWORK
TITLE =

      A     DB10.DBX   61.2;
      =     DB3.DBX    3.7;
NETWORK
TITLE =

      A     M    182.0;
      =     DB3.DBX    2.0;
NETWORK
TITLE =

      A     M    183.0;
      =     DB3.DBX    2.1;
NETWORK
TITLE =

      A     M    208.0;
      =     DB3.DBX    2.2;
NETWORK
TITLE =

      A     M    212.0;
      =     DB3.DBX    2.3;
NETWORK
TITLE =
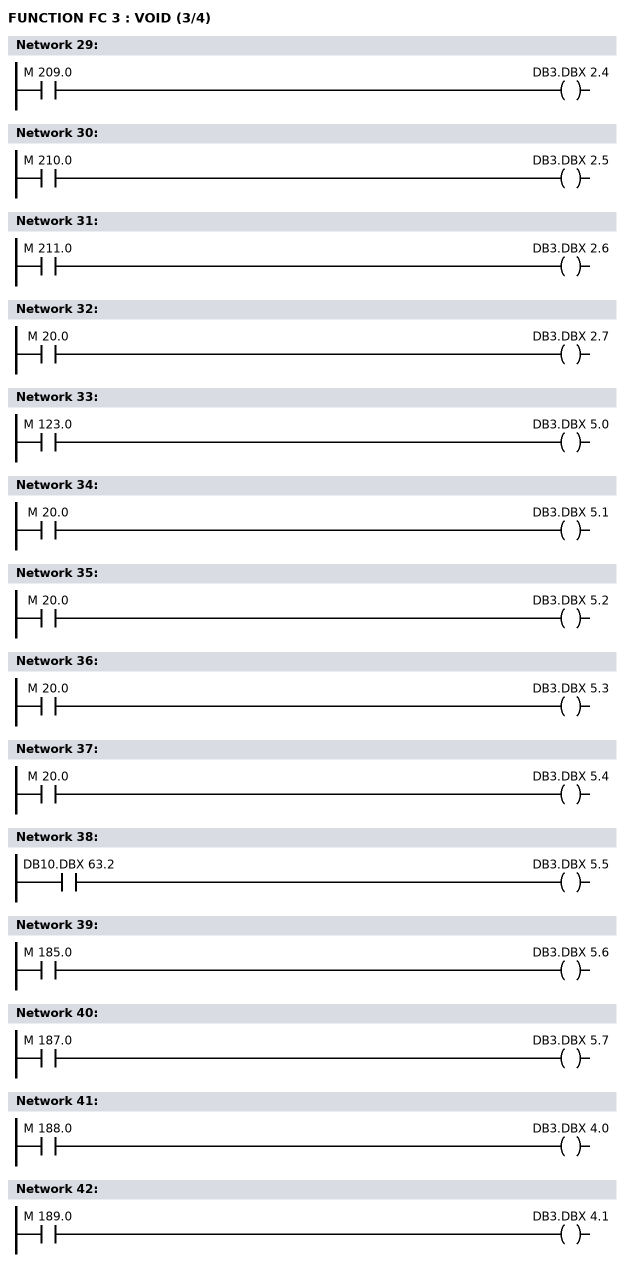

      A     M    209.0;
      =     DB3.DBX    2.4;
NETWORK
TITLE =

      A     M    210.0;
      =     DB3.DBX    2.5;
NETWORK
TITLE =

      A     M    211.0;
      =     DB3.DBX    2.6;
NETWORK
TITLE =

      A     M     20.0;
      =     DB3.DBX    2.7;
NETWORK
TITLE =

      A     M    123.0;
      =     DB3.DBX    5.0;
NETWORK
TITLE =

      A     M     20.0;
      =     DB3.DBX    5.1;
NETWORK
TITLE =

      A     M     20.0;
      =     DB3.DBX    5.2;
NETWORK
TITLE =

      A     M     20.0;
      =     DB3.DBX    5.3;
NETWORK
TITLE =

      A     M     20.0;
      =     DB3.DBX    5.4;
NETWORK
TITLE =

      A     DB10.DBX   63.2;
      =     DB3.DBX    5.5;
NETWORK
TITLE =

      A     M    185.0;
      =     DB3.DBX    5.6;
NETWORK
TITLE =

      A     M    187.0;
      =     DB3.DBX    5.7;
NETWORK
TITLE =

      A     M    188.0;
      =     DB3.DBX    4.0;
NETWORK
TITLE =

      A     M    189.0;
      =     DB3.DBX    4.1;
NETWORK
TITLE =
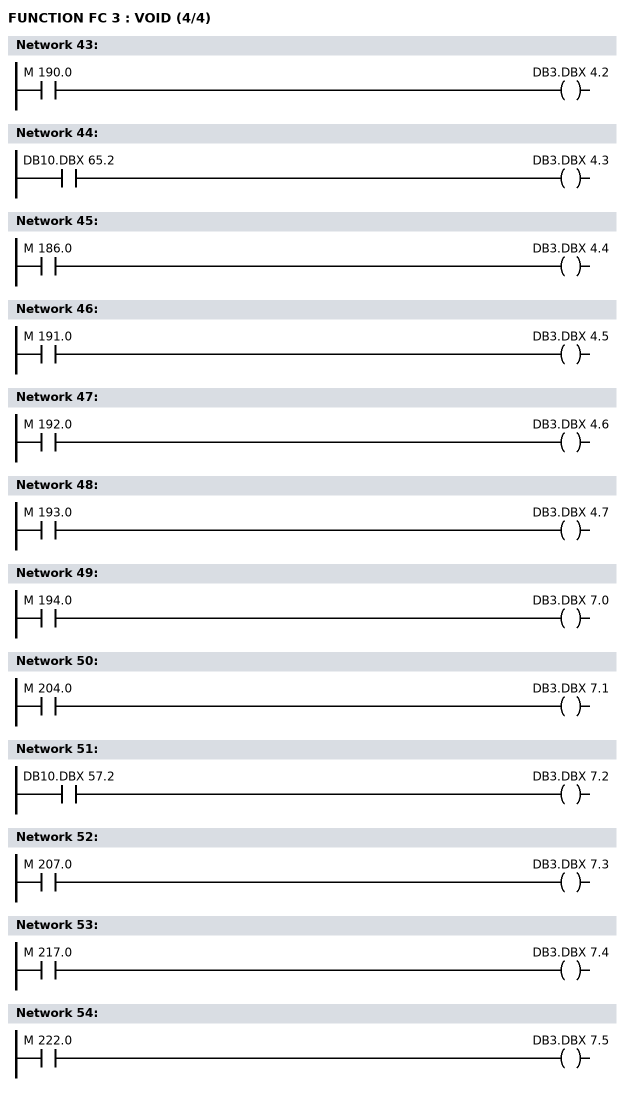

      A     M    190.0;
      =     DB3.DBX    4.2;
NETWORK
TITLE =

      A     DB10.DBX   65.2;
      =     DB3.DBX    4.3;
NETWORK
TITLE =

      A     M    186.0;
      =     DB3.DBX    4.4;
NETWORK
TITLE =

      A     M    191.0;
      =     DB3.DBX    4.5;
NETWORK
TITLE =

      A     M    192.0;
      =     DB3.DBX    4.6;
NETWORK
TITLE =

      A     M    193.0;
      =     DB3.DBX    4.7;
NETWORK
TITLE =

      A     M    194.0;
      =     DB3.DBX    7.0;
NETWORK
TITLE =

      A     M    204.0;
      =     DB3.DBX    7.1;
NETWORK
TITLE =

      A     DB10.DBX   57.2;
      =     DB3.DBX    7.2;
NETWORK
TITLE =

      A     M    207.0;
      =     DB3.DBX    7.3;
NETWORK
TITLE =

      A     M    217.0;
      =     DB3.DBX    7.4;
NETWORK
TITLE =

      A     M    222.0;
      =     DB3.DBX    7.5;
END_FUNCTION

FUNCTION FC 10 : VOID
AUTHOR :
FAMILY : GENERAL
NAME : GENERAL
VERSION : 0.0


VAR_TEMP
  TEMP0 : BOOL ;
  TEMP1 : BOOL ;
  TEMP2 : BOOL ;
  TEMP3 : BOOL ;
END_VAR
BEGIN
NETWORK
TITLE =
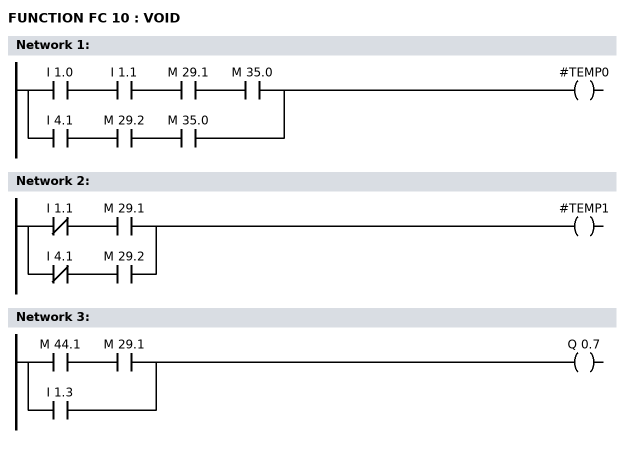

      A     I      1.0;
      A     I      1.1;
      A     M     29.1;
      A     M     35.0;
      O     ;
      A     I      4.1;
      A     M     29.2;
      A     M     35.0;
      =     #TEMP0;
NETWORK
TITLE =

      AN    I      1.1;
      A     M     29.1;
      O     ;
      AN    I      4.1;
      A     M     29.2;
      =     #TEMP1;
NETWORK
TITLE =

      A     M     44.1;
      A     M     29.1;
      O     I      1.3;
      =     Q      0.7;
NETWORK
TITLE =

      A(    ;
      O     M     29.1;
      O     M     29.0;
      O     ;
      A(    ;
      A     I      4.6;
      L     S5T#2M;
      SF    T     46;
      NOP   0;
      NOP   0;
      NOP   0;
      A     T     46;
      )     ;
      A     M     29.2;
      O     I      4.2;
      )     ;
      AN    M    114.0;
      AN    M    207.0;
      AN    M    206.0;
      AN    M    167.0;
      AN    M    206.0;
      AN    M    207.0;
      A     I     10.3;
      AN    M    209.0;
      AN    M    210.0;
      AN    M    211.0;
      A     M    121.7;
      AN    M    122.1;
      AN    M    123.0;
      AN    M    155.0;
      AN    M    158.0;
      AN    M    166.0;
      AN    M    175.0;
      AN    M    179.0;
      AN    M    208.0;
      AN    M    163.4;
      AN    M    212.0;
      A(    ;
      A     M      0.1;
      AN    I      4.3;
      O     ;
      A     M      0.2;
      AN    I      4.4;
      )     ;
      A     M    150.5;
      A     M    150.6;
      AN    M    151.0;
      AN    M    180.0;
      A(    ;
      A     Q      6.0;
      AN    I      8.3;
      NOT   ;
      )     ;
      =     M     35.1;
NETWORK
TITLE =
